// ---- Data types/Beckhoff IO udts/udt_EP2328_0002.TcDUT
(*udt (user defined type) of Beckhoff EP2028-0002 - 8 Point IP67 Rated Digital Output Box:
	auth. Brent Lekx-Toniolo of Toniolo Research & Development Inc.; 
	July 2010;
	Modified for tag reduction by R.Remillard
	November 2012; version 2.0*)


TYPE udt_EP2328_0002 :
STRUCT
	Q AT %Q*: BYTE;
	I AT %I*: BYTE;
	
	(*Status bits*)
	WC_State AT %I*:BOOL;
	State AT %I*: UINT;

END_STRUCT
END_TYPE

// ---- Data types/Beckhoff IO udts/udt_EP2624.TcDUT
(*udt (user defined type) of Beckhoff EL2624 - 4 Point Relay Type Output Terminal:
	Auth: j.vandongen
	October 2019*)


TYPE udt_EP2624 :
STRUCT
	Q: INT;
END_STRUCT
END_TYPE

// ---- Data types/Beckhoff IO udts/udt_EP2624_STAT.TcDUT
(*udt (user defined type) of Beckhoff EL2624 - 4 Point Relay Type Output Terminal:
	Auth: j.vandongen
	October 2019*)


TYPE udt_EP2624_STAT :
STRUCT
	InfoData: udt_ECATSlave_Status;
END_STRUCT
END_TYPE

// ---- Data types/Beckhoff IO udts/udt_EP3174_0002.TcDUT
(*udt (user defined type) of Beckhoff EP3174_0002 - 4 channel,  Analog Input Terminal:*)


TYPE udt_EP3174_0002 :
STRUCT

	CH1: INT;
	CH2: INT;
	CH3: INT;
	CH4: INT;
	InfoData: udt_ECATSlave_Status;

END_STRUCT
END_TYPE

// ---- Data types/Beckhoff IO udts/udt_EP6224.TcDUT
(*udt (user defined type) of Beckhoff EP6224-0002 - 4 Point IP67 Rated IO-Link Box:
	Version 20190506
		- initial creation, j.vandongen


*)


TYPE udt_EP6224 :
STRUCT

	Device_Diag: BOOL;
	Device_Stat: BOOL;


(* DeviceState Inputs:
	0x_0 = Port disabled
	0x_1 = Port in std dig in
	0x_2 = Port in std dig out
	0x_3 = Port in communikation OP
	0x_4 = Port in communikation COMSTOP
	0x1_ = Watchdog detected
	0x2_ = internal Error
	0x3_ = invalid Device ID
	0x4_ = invalid Vendor ID
	0x5_ = invalid IO-Link Version
	0x6_ = invalid Frame Capability
	0x7_ = invalid Cycle Time
	0x8_ = invalid PD in length
	0x9_ = invalid PD out length
	0xA_ = no Device detected
	0xB_ = error Preoperate
*)
	State_Ch1: USINT;
	State_Ch2: USINT;
	State_Ch3: USINT;
	State_Ch4: USINT;


	Port1_ProcessData: ARRAY [0..7] OF USINT;
	Port2_ProcessData: ARRAY [0..7] OF USINT;
	Port3_ProcessData: ARRAY [0..7] OF USINT;
	Port4_ProcessData: ARRAY [0..7] OF USINT;


	InfoData: udt_ECATSlave_StatusADS;

END_STRUCT
END_TYPE

// ---- Data types/Beckhoff IO udts/udt_EP6224_CMD.TcDUT
(*udt (user defined type) of Beckhoff EP6224-0002 - 4 Point IP67 Rated IO-Link Box:
	Version 20190506
		- initial creation, j.vandongen


*)


TYPE udt_EP6224_CMD :
STRUCT
	Port1_Q: BOOL;
	Port2_Q: BOOL;
	Port3_Q: BOOL;
	Port4_Q: BOOL;

END_STRUCT
END_TYPE

// ---- Data types/Beckhoff IO udts/udt_EP6224_I.TcDUT
(*udt (user defined type) of Beckhoff EP6224-0002 - 4 Point IP67 Rated IO-Link Box:
	Version 20210621
		- initial creation, j.underhill

*)


TYPE udt_EP6224_I :
STRUCT
	Port1_I: BOOL;
	Port2_I: BOOL;
	Port3_I: BOOL;
	Port4_I: BOOL;

END_STRUCT
END_TYPE

// ---- Data types/Beckhoff IO udts/udt_EP9128_20250704.TcDUT
(*udt (user defined type) of Beckhoff CU1128 - EtherCAT Junction:
	
------------------------------------------------------------------------
REVISION NOTES:
	Original Author(s): b.lekx-toniolo, copied from CU1128: r.jones
	Version 20250704
		- Initial Concept

------------------------------------------------------------------------
*)
TYPE udt_EP9128_20250704 :
STRUCT
	InfoData: udt_ECATSlave_Status_EP9128;
	InfoDataB: udt_ECATSlave_Status_EP9128;
	InfoDataC: udt_ECATSlave_Status_EP9128;
END_STRUCT
END_TYPE

// ---- Data types/Beckhoff IO udts/udt_EP9214_CH_CMD_20250704.TcDUT
(*udt (user defined type) of Beckhoff EP9214 IP67 Block - Power Distribution Block, individual channel data:
	To work in conjunction of udt_EP9214_STAT_yyyymmdd
	auth. Brent Lekx-Toniolo, copy/paste from 9224 from r.jones of Sodecia GTAC; 

------------------------------------------------------------------------
REVISION NOTES:
	Version 20250704
		- Initial Concept
------------------------------------------------------------------------

*)


TYPE udt_EP9214_CH_CMD_20250704 :
STRUCT

	Output_Us: BOOL;
	Output_Up: BOOL;
	Reset_Us: BOOL;
	Reset_Up: BOOL;

END_STRUCT
END_TYPE

// ---- Data types/Beckhoff IO udts/udt_EP9214_CH_STAT_20250704.TcDUT
(*udt (user defined type) of Beckhoff EP9214 IP67 Block - Power Distribution Block, individual channel data:
	To work in conjunction of udt_EP9214_STAT_yyyymmdd
	auth. Brent Lekx-Toniolo, copy/paste from 9224 from r.jones of Sodecia GTAC; 

------------------------------------------------------------------------
REVISION NOTES:
	Version 20250704
		- Initial Concept
------------------------------------------------------------------------

*)


TYPE udt_EP9214_CH_STAT_20250704 :
STRUCT

	Error_Us: BOOL;
	Error_Up: BOOL;
	Warning_Us: BOOL;
	Warning_Up: BOOL;
	Status_Us: BOOL;
	Status_Up: BOOL;
	Channel_Error: BOOL;
	SyncError: BOOL;
	TxPDO_State: BOOL;
	TxPDO_Toggle: BOOL;

END_STRUCT
END_TYPE

// ---- Data types/Beckhoff IO udts/udt_EP9214_CMD_20250704.TcDUT
(*udt (user defined type) of Beckhoff EP9214 IP67 Block - Power Distribution Block, individual channel data:
	To work in conjunction of udt_EP9214_STAT_yyyymmdd
	auth. Brent Lekx-Toniolo, copy/paste from 9224 from r.jones of Sodecia GTAC; 

------------------------------------------------------------------------
REVISION NOTES:
	Version 20250704
		- Initial Concept
------------------------------------------------------------------------
------------------------------------------------------------------------
*)
TYPE udt_EP9214_CMD_20250704 :
STRUCT

	(*Channel Specific Commands*)
	Channel1: udt_EP9214_CH_CMD_20250704;
	Channel2: udt_EP9214_CH_CMD_20250704;
	Channel3: udt_EP9214_CH_CMD_20250704;
	Channel4: udt_EP9214_CH_CMD_20250704;

	(*Overall Device Commands*)
	Device: udt_EP9214_DEV_CMD_20250704;

END_STRUCT
END_TYPE

// ---- Data types/Beckhoff IO udts/udt_EP9214_DEV_CMD_20250704.TcDUT
(*udt (user defined type) of Beckhoff EP9214 IP67 Block - Power Distribution Block, individual channel data:
	To work in conjunction of udt_EP9214_STAT_yyyymmdd
	auth. Brent Lekx-Toniolo, copy/paste from 9224 from r.jones of Sodecia GTAC; 

------------------------------------------------------------------------
REVISION NOTES:
	Version 20250704
		- Initial Concept
------------------------------------------------------------------------

*)


TYPE udt_EP9214_DEV_CMD_20250704 :
STRUCT

	Enable_Control_Via_Fieldbus: BOOL;
	Global_Reset: BOOL;

END_STRUCT
END_TYPE

// ---- Data types/Beckhoff IO udts/udt_EP9214_DEV_STAT_20250704.TcDUT
(*udt (user defined type) of Beckhoff EP9214 IP67 Block - Power Distribution Block, individual channel data:
	To work in conjunction of udt_EP9214_STAT_yyyymmdd
	auth. Brent Lekx-Toniolo, copy/paste from 9224 from r.jones of Sodecia GTAC; 

------------------------------------------------------------------------
REVISION NOTES:
	Version 20250704
		- Initial Concept
------------------------------------------------------------------------

*)


TYPE udt_EP9214_DEV_STAT_20250704 :
STRUCT

	Temperature_Warning: BOOL;
	Temperature_Error: BOOL;
	Us_Warning: BOOL;
	Us_Error: BOOL;
	Up_Warning: BOOL;
	Up_Error: BOOL;
	Global_Error_Bit: BOOL;
	Reset_Input: BOOL;
	TxPDO_State: BOOL;
	TxPDO_Toggle: BOOL;

END_STRUCT
END_TYPE

// ---- Data types/Beckhoff IO udts/udt_EP9214_STAT_20250704.TcDUT
(*udt (user defined type) of Beckhoff EP9214 IP67 Block - Power Distribution Block, individual channel data:
	To work in conjunction of udt_EP9214_STAT_yyyymmdd
	auth. Brent Lekx-Toniolo, copy/paste from 9224 from r.jones of Sodecia GTAC; 

------------------------------------------------------------------------
REVISION NOTES:
	Version 20250704
		- Initial Concept
------------------------------------------------------------------------

*)


TYPE udt_EP9214_STAT_20250704 :
STRUCT

	(*Channel Specific Status*)
	Channel_1: udt_EP9214_CH_STAT_20250704;
	Channel_2: udt_EP9214_CH_STAT_20250704;
	Channel_3: udt_EP9214_CH_STAT_20250704;
	Channel_4: udt_EP9214_CH_STAT_20250704;

	(*Overall Device Status*)
	Device: udt_EP9214_DEV_STAT_20250704;


	(*EtherCAT Slave Status*)
	Wc_State: BOOL;
	(*0 = Data valid
	1 = Data invalid*)
	InfoData: udt_ECATSlave_StatusEXT;

END_STRUCT
END_TYPE

// ---- Data types/Beckhoff IO udts/udt_EP9224_CH_CMD_20161207.TcDUT
(*udt (user defined type) of Beckhoff EP9224 IP67 Block - Power Distribution Block, individual channel commands
	To work in conjunction of udt_EP9224_CMDyymmdd
	auth. Brent Lekx-Toniolo of Sodecia GTAC; 

------------------------------------------------------------------------
REVISION NOTES:
	Version 20161207
		- Initial Concept
------------------------------------------------------------------------

*)


TYPE udt_EP9224_CH_CMD_20161207 :
STRUCT

	Output_Us: BOOL;
	Output_Up: BOOL;
	Reset_Us: BOOL;
	Reset_Up: BOOL;

END_STRUCT
END_TYPE

// ---- Data types/Beckhoff IO udts/udt_EP9224_CH_STAT_20161207.TcDUT
(*udt (user defined type) of Beckhoff EP9224 IP67 Block - Power Distribution Block, individual channel data:
	To work in conjunction of udt_EP9224_STAT_yyyymmdd
	auth. Brent Lekx-Toniolo of Sodecia GTAC; 

------------------------------------------------------------------------
REVISION NOTES:
	Version 20161207
		- Initial Concept
------------------------------------------------------------------------

*)


TYPE udt_EP9224_CH_STAT_20161207 :
STRUCT

	Error_Us: BOOL;
	Error_Up: BOOL;
	Warning_Us: BOOL;
	Warning_Up: BOOL;
	Status_Us: BOOL;
	Status_Up: BOOL;
	Channel_Error: BOOL;
	Error_Sum_Current: BOOL;
	Warning_Sum_Current: BOOL;
	TxPDO_State: BOOL;
	TxPDO_Toggle: BOOL;
	Current_Us: INT;
	Current_Up: INT;

END_STRUCT
END_TYPE

// ---- Data types/Beckhoff IO udts/udt_EP9224_CMD_20161207.TcDUT
(*udt (user defined type) of Beckhoff EP9224 IP67 Block - Power Distribution Block:
	To work in conjunction of udt_EP9224_STAT_yyyymmdd
	auth. Brent Lekx-Toniolo of Sodecia GTAC; 


------------------------------------------------------------------------
REVISION NOTES:
	Version 20161207
		- Initial Concept
------------------------------------------------------------------------
*)
TYPE udt_EP9224_CMD_20161207 :
STRUCT

	(*Channel Specific Commands*)
	Channel1: udt_EP9224_CH_CMD_20161207;
	Channel2: udt_EP9224_CH_CMD_20161207;
	Channel3: udt_EP9224_CH_CMD_20161207;
	Channel4: udt_EP9224_CH_CMD_20161207;

	(*Overall Device Commands*)
	Device: udt_EP9224_DEV_CMD_20161207;

END_STRUCT
END_TYPE

// ---- Data types/Beckhoff IO udts/udt_EP9224_DEV_CMD_20161207.TcDUT
(*udt (user defined type) of Beckhoff EP9224 IP67 Block - Power Distribution Block, device commands
	To work in conjunction of udt_EP9224_CMDyymmdd
	auth. Brent Lekx-Toniolo of Sodecia GTAC; 

------------------------------------------------------------------------
REVISION NOTES:
	Version 20161207
		- Initial Concept
------------------------------------------------------------------------

*)


TYPE udt_EP9224_DEV_CMD_20161207 :
STRUCT

	Enable_Control_Via_Fieldbus: BOOL;
	Global_Reset: BOOL;

END_STRUCT
END_TYPE

// ---- Data types/Beckhoff IO udts/udt_EP9224_DEV_STAT_20161207.TcDUT
(*udt (user defined type) of Beckhoff EP9224 IP67 Block - Power Distribution Block, device data:
	To work in conjunction of udt_EP9224_STAT_yyyymmdd
	auth. Brent Lekx-Toniolo of Sodecia GTAC; 

------------------------------------------------------------------------
REVISION NOTES:
	Version 20161207
		- Initial Concept
------------------------------------------------------------------------

*)


TYPE udt_EP9224_DEV_STAT_20161207 :
STRUCT

	Temperature_Warning: BOOL;
	Temperature_Error: BOOL;
	Us_Warning: BOOL;
	Us_Error: BOOL;
	Up_Warning: BOOL;
	Up_Error: BOOL;
	Global_Error_Bit: BOOL;
	Sum_Curent_Warning: BOOL;
	Sum_Current_Error: BOOL;
	Reset_Input: BOOL;
	TxPDO_State: BOOL;
	TxPDO_Toggle: BOOL;
	Current_Us: INT;
	Current_Up: INT;
	Voltage_Us: INT;
	Voltage_Up: INT;
	Temperature: INT;

END_STRUCT
END_TYPE

// ---- Data types/Beckhoff IO udts/udt_EP9224_STAT_20161207.TcDUT
(*udt (user defined type) of Beckhoff EP9224 IP67 Block - Power Distribution Block:
	To work in conjunction of udt_EP9224_yyyymmdd
	auth. Brent Lekx-Toniolo of Sodecia GTAC; 

------------------------------------------------------------------------
REVISION NOTES:
	Version 20161207
		- Initial Concept
------------------------------------------------------------------------

*)


TYPE udt_EP9224_STAT_20161207 :
STRUCT

	(*Channel Specific Status*)
	Channel_1: udt_EP9224_CH_STAT_20161207;
	Channel_2: udt_EP9224_CH_STAT_20161207;
	Channel_3: udt_EP9224_CH_STAT_20161207;
	Channel_4: udt_EP9224_CH_STAT_20161207;

	(*Overall Device Status*)
	Device: udt_EP9224_DEV_STAT_20161207;


	(*EtherCAT Slave Status*)
	Wc_State: BOOL;
	(*0 = Data valid
	1 = Data invalid*)
	InfoData: udt_ECATSlave_StatusEXT;

END_STRUCT
END_TYPE

// ---- Data types/Beckhoff IO udts/udt_ProfiMaster_Status.TcDUT
(*udt (user defined type) of Generic Profibus Master to Store Data for Status of any Profibus Master Modules:
	auth. brent lekx-toniolo; April 2008*)

TYPE udt_ProfiMaster_Status :
	STRUCT
		(*CdlInfo*)
		cycleCounter: UINT;
		error: USINT;
		actualCycleTime: UINT;
		actualModulo: USINT;
		(*CycleCounter:
  			FCxxxx increments this counter once after each cycle
		Error:
  			indicates the number of boxes with a BoxState unequal zero
		ActualCycleTime:
  			indicates the actual Cycle-Time (in 4/25 µs)
		ActualModulo:
  			indicates the actual Modulo in case of different poll cycles of the boxes*)

		(*Counter*)
		Counter0: UINT;
		Counter1: UINT;
		Counter2: UINT;
		Counter3: UINT;
		Counter4: UINT;
		Counter5: UINT;
		Counter6: UINT;
		Counter7: UINT;
		(*	Counter[0-1]: reserved for future
			Counter[2]: ReceivedTelegram-Counter (in Redundancy Mode)
  				FCxxxx increments this counter once every time when a correct
  				PROFIBUS-telegram is received (only in Redundancy Mode)
			Counter[3]: ReceivedTelegramFromPrimaryMaster-Counter (in Redundancy Mode)
  				FCxxxx increments this counter once every time when a correct
  				PROFIBUS-telegram from the Primary Master (which has the same
  				station address as the Redundancy Master is received (only in Redundancy Mode)
			Counter[4]: ClaimTokenTimeout-Counter (in Redundancy Mode)
  				FCxxxx increments this counter once every time when a Timeout on the
  				PROFIBUS occurs (only in Redundancy Mode)
			Counter[5-7]: reserved for future*)

		DiagFlag: BOOL;

		(*GlobalState*)
		GlobalState0: UINT;
		GlobalState1: UINT;
		GlobalState2: UINT;
		GlobalState3: UINT;
			(*GlobalState[0]:
  				0: FC310x is in state RUN
  				1: FC310x is in state RESET
  				2: FC310x is in state OFFLINE
  				3: FC310x is in state STOP
			GlobalState[1]:
  				number of bus errors detected
			GlobalState[2]:
  				reserved for future use*)

		LastAdsError: UINT;
		CycleFailedCounter: UINT;
	END_STRUCT

END_TYPE

// ---- Data types/Beckhoff IO udts/udt_ProfiNet_Status.TcDUT
TYPE udt_ProfiNet_Status :
STRUCT
	
	PnIoBoxState : UINT;
(*
0 = No error
1 = Profinet device state machine is in boot mode
2 = Device not found
3 = The stationname is not unique
4 = IP could not be set
5 = IP conflict
6 = DCP set was not successful
7 = Watchdog error
8 = Datahold error
9 = RTC3: Sync mode could not be initiated
10 = Profinet controller has a link error
11 = The aliasname is not unique
12 = The automatic name assignement isn't possible - wrong device type
13 = IOC-AR is established but no application ready
14 = IOC-AR is established but module difference
15 = At least one InputCR is invalid, provider in stop or problemindicator is set
16 = At least one OutputCR is invalid, provider in stop or problemindicator is set
31 = Only for EtherCAT gateways: WC-State of cyclic EtherCAT frame is 1
*)

END_STRUCT
END_TYPE

// ---- Data types/Beckhoff IO udts/udt_ProfiNode_Status.TcDUT
(*udt (user data type) of Generic Profibus Node to Store Data for Status of any Profibus Modules:
	auth. brent lekx-toniolo; April 2008
	version 1.0*)


TYPE udt_ProfiNode_Status :
	STRUCT
		DpState: USINT;
		(*0 = No error
		1 = Station deactivated
		2 = Station not exists
		3 = Master lock
		4 = Invalid slave response
		5 = Parameter fault
		6 = Not supported
		7 = Config fault
		8 = Station not ready
		9 = Static diagnosis
		10 = Diagnosis overflow
		11 = Physical fault
		12 = Data-Exchange left
		13 = Severe bus fault
		14 = Telegram fault
		15 = Station has no ressources
		16 = Service not activated
		17 = Unexpected telegram
		18 = Station ready
		128 = slave, waiting for data transfer
		129	= slave, waiting for configuration
		130	= slave, waiting for parameter*)
		ExtDiagFlag: BOOL;

	END_STRUCT
END_TYPE

// ---- Data types/Beckhoff IO udts/udt_SMB_Status_20141211.TcDUT
(*udt used to create memory space for linking to SMB diagnositcs
For use with Motherboards that contain LM75 and/or LM78 chips accessed via System Management Bus (SMB)


------------------------------------------------------------------------
REVISION NOTES:
	Original Author(s): b.lekx-toniolo, JVD, Chris Timmermans (Edge)
	Version 20141211
		- First Draft

------------------------------------------------------------------------
*)




TYPE udt_SMB_Status_20141211 :
STRUCT
	Temp_MB: 	UINT; 		(*°C*)
	Fan_0: 		UINT;		(*RPM*)
	Fan_1: 		UINT;		(*RPM*)
	Fan_2: 		UINT;		(*RPM*)
	Volt_2a: 		UINT;		(*0.01V*)
	Volt_2b: 		UINT;		(*0.01V*)
	Volt_33: 		UINT;		(*0.01V*)
	Volt_5: 		UINT;		(*0.01V*)
	Volt_12: 		UINT;		(*0.01V*)
	Volt_neg12: 	UINT;		(*0.01V*)
	Volt_neg5: 	UINT;		(*0.01V*)
	Temp_0: 	USINT;		(*°C*)
	Temp_1: 	USINT;		(*°C*)
	Temp_2: 	USINT;		(*°C*)
	Temp_3: 	USINT;		(*°C*)
	Temp_4: 	USINT;		(*°C*)
	Temp_5: 	USINT;		(*°C*)
	Temp_6:		USINT;		(*°C*)
	Temp_7: 	USINT;		(*°C*)


END_STRUCT
END_TYPE

// ---- Data types/Discrete Image udts/udt_ATIxx_Image_20151104.TcDUT
(*udt (user defined type) for all generic ATI Tool changers
	auth. Brent Lekx-Toniolo of Sodecia GTAC

------------------------------------------------------------------------
REVISION NOTES:

	Version 20151104:
	- initial concept, b.lekx-toniolo	
------------------------------------------------------------------------

*)

TYPE udt_ATIxx_Image_20151104 :
	STRUCT
			(*Input Data Image*)
			In_From_Hardware: udt_ATI_Input_20150203;
			(*Output Data Image*)
			Out_To_Hardware: udt_ATI_Output_20150203;

			(*Cable Break States*)
			ECatSlave_Cable_Breaks: UDINT;

	END_STRUCT
END_TYPE

// ---- Data types/Discrete Image udts/udt_Drive_Image_20160804.TcDUT
(*udt (user defined type) of Beckhoff Type for Storage of Visualization for Servo Drive Data
	auth. Brent Lekx-Toniolo of Toniolo Research & Development Inc.; 
	SORT OF RUSHED!!!
	Sept 2010; version 1.0

	Version 1.0: Sept2010
		- Initial Concept
	Version 1.1
		- A little less RUSHED, r.remillard
	Version 1.2
		- Added extra var for error April 21 2015 Chris Timmermans
	Version20160804
		- Changed Name for convention, b.lekx-toniolo
		- Moved Safety Diag and Safety Status Words from UI section to this udt, b.lekx-toniolo
		- Created Arrays for Multi axis use per drive system, b.lekx-toniolo
		- Added Seperated Error IDs and Strings, b.lekx-toniolo
*)



TYPE udt_Drive_Image_20160804 :
	STRUCT
	(*General Status of Drive SYSTEM and FB*)
	In_Play_ACK: ARRAY[1..2] OF BOOL;
	In_Teach_ACK: ARRAY[1..2] OF BOOL;
	Homed: ARRAY[1..2] OF BOOL;
	In_Motion: ARRAY[1..2] OF BOOL;
	In_Requested_Position: ARRAY[1..2] OF BOOL;
	Current_Step_Pointer: ARRAY[1..2] OF UDINT;
	At_Current_Step: ARRAY[1..2] OF UINT;
	Prev_Step_Data: ARRAY[1..2] OF udt_SingleAxis_MoveData_20160908;
	Current_Step_Data: ARRAY[1..2] OF udt_SingleAxis_MoveData_20160908;
	Next_Step_Data: ARRAY[1..2] OF udt_SingleAxis_MoveData_20160908;
	Cycle_Complete: ARRAY[1..2] OF BOOL;

	(*Status of Physical Drive Unit and Axis*)
	AX5xxx: udt_AX5206_20160804;
	EL7xxx: udt_EL7211_20150115;

	AX5805: udt_AX5805_20160804;
	Safety_DIAG: 	udt_AX5805_DiagData;
	Safety_STAT: DINT;

	Drive_Type_Message: ARRAY[1..2] OF STRING;
	Drive_OperationalState: ARRAY[1..2] OF E_AX5000_DriveOpMode;

	Drive_In_Error: ARRAY[1..2] OF BOOL;
	Drive_Status: ARRAY[1..2] OF UINT;
	Drive_StatusStruct: ARRAY[1..2] OF ST_AX5000DriveStatus;
	Drive_Status_Message: ARRAY[1..2] OF STRING;
	Drive_Diag_ErrorID: ARRAY[1..2] OF UDINT;
	Drive_Diag_Message: ARRAY[1..2] OF STRING;
	Drive_C1D_ErrorID: ARRAY[1..2] OF UINT;
	Drive_C1D_ErrorStruct: ARRAY [1..2] OF ST_AX5000_C1D;
	Drive_C1D_Error_Message: ARRAY[1..2] OF STRING;

	Axis_Motor_Message: ARRAY[1..2] OF STRING;
	Axis_In_Error: ARRAY[1..2] OF BOOL;
	Axis_ErrorID: ARRAY[1..2] OF DWORD;
	Axis_ErrorMessage: ARRAY[1..2] OF STRING;

	Actual_Position: ARRAY[1..2] OF LREAL;
	Software_Limit_Exceeded: ARRAY[1..2]OF BOOL;
	Is_Calibrated: ARRAY[1..2] OF BOOL;
	StateDWord: ARRAY[1..2] OF DWORD;
	Ready: ARRAY[1..2] OF BOOL;



	END_STRUCT
END_TYPE

// ---- Data types/Discrete Image udts/udt_Drive_Image_20190816.TcDUT
(*udt (user defined type) of Beckhoff Type for Storage of Visualization for Servo Drive Data
	auth. Brent Lekx-Toniolo of Toniolo Research & Development Inc.; 
	SORT OF RUSHED!!!
	Sept 2010; version 1.0

	Version 1.0: Sept2010
		- Initial Concept
	Version 1.1
		- A little less RUSHED, r.remillard
	Version 1.2
		- Added extra var for error April 21 2015 Chris Timmermans
	Version20160804
		- Changed Name for convention, b.lekx-toniolo
		- Moved Safety Diag and Safety Status Words from UI section to this udt, b.lekx-toniolo
		- Created Arrays for Multi axis use per drive system, b.lekx-toniolo
		- Added Seperated Error IDs and Strings, b.lekx-toniolo
		- Added Axis ID Strings, b.lekx-toniolo
	Version 20180801
		- teach enabled added, b.donnell 
	Version 20190816
		-added "Corrected Positon" var for crankshaft/coupling conversions for UI displaying purposes, j.underhill (Fork Drilling Machine)
*)



TYPE udt_Drive_Image_20190816 :
	STRUCT

	(*Identification String for general purpose UI*)
	Axis_Common_Name: ARRAY[0..2] OF STRING[30];

	(*General Status of Drive SYSTEM and FB*)
	In_Play_ACK: ARRAY[0..2] OF BOOL;
	In_Teach_ACK: ARRAY[0..2] OF BOOL;
	Homed: ARRAY[0..2] OF BOOL;
	In_Motion: ARRAY[0..2] OF BOOL;
	In_Requested_Position: ARRAY[0..2] OF BOOL;
	Current_Step_Pointer: ARRAY[0..2] OF UDINT;
	At_Current_Step: ARRAY[0..2] OF UINT;
	Prev_Step_Data: ARRAY[0..2] OF udt_SingleAxis_MoveData_20160908;
	Current_Step_Data: ARRAY[0..2] OF udt_SingleAxis_MoveData_20160908;
	Next_Step_Data: ARRAY[0..2] OF udt_SingleAxis_MoveData_20160908;
	Cycle_Complete: ARRAY[0..2] OF BOOL;
	Teach_Enable: ARRAY[0..2] OF BOOL;

	(*Status of Physical Drive Unit and Axis*)
	AX5xxx: udt_AX5206_20160804;
	EL7xxx: udt_EL7211_20150115;

	AX5805: udt_AX5805_20160804;
	Safety_DIAG: 	udt_AX5805_DiagData;
	Safety_STAT: DINT;

	Drive_Type_Message: ARRAY[0..2] OF STRING;
	Drive_OperationalState: ARRAY[0..2] OF E_AX5000_DriveOpMode;

	Drive_In_Error: ARRAY[0..2] OF BOOL;
	Drive_Status: ARRAY[0..2] OF UINT;
	Drive_StatusStruct: ARRAY[0..2] OF ST_AX5000DriveStatus;
	Drive_Status_Message: ARRAY[0..2] OF STRING;
	Drive_Diag_ErrorID: ARRAY[0..2] OF UDINT;
	Drive_Diag_Message: ARRAY[0..2] OF STRING;
	Drive_C1D_ErrorID: ARRAY[0..2] OF UINT;
	Drive_C1D_ErrorStruct: ARRAY [0..2] OF ST_AX5000_C1D;
	Drive_C1D_Error_Message: ARRAY[0..2] OF STRING;

	Axis_Motor_Message: ARRAY[0..2] OF STRING;
	Axis_In_Error: ARRAY[0..2] OF BOOL;
	Axis_ErrorID: ARRAY[0..2] OF DWORD;
	Axis_ErrorMessage: ARRAY[0..2] OF STRING;

	Corrected_Position: ARRAY[0..2] OF LREAL;
	Actual_Position: ARRAY[0..2] OF LREAL;
	Software_Limit_Exceeded: ARRAY[0..2]OF BOOL;
	Is_Calibrated: ARRAY[0..2] OF BOOL;
	StateDWord: ARRAY[0..2] OF DWORD;
	Ready: ARRAY[0..2] OF BOOL;



	END_STRUCT
END_TYPE

// ---- Data types/Discrete Image udts/udt_ECATMaster_Image_20220224.TcDUT
(*udt (user defined type) for full display (By GTAC Standards) of EtherCAT Master:
	auth. Brent Lekx-Toniolo of Toniolo Research & Development Inc.; 
	Version 20160407
		- initial concept, b.lekx-toniolo
	Version 20220224
	- Change Config array start element from 1 to 0 for TcUI migration project, b.lekx-toniolo / c.drees

*)



TYPE udt_ECATMaster_Image_20220224 :
STRUCT
	HW: udt_ECATMaster_Status_20141211;
	AMS_ID: STRING;
	Config: ARRAY [0..100] OF STRING[5];


END_STRUCT
END_TYPE

// ---- Data types/Discrete Image udts/udt_ECATNodeConfig_20200729.TcDUT
TYPE udt_ECATNodeConfig_20200729 :
STRUCT
		FixtureConfig:ARRAY [0..120] OF udt_ECATNodeData_20221507;								(*Storage Area for Actual GTAC Fixture Device Based Config*)
		EOATConfig:ARRAY[0..15] OF udt_ECATNodeData_20221507;
		ATIConfig:ARRAY[0..5] OF udt_ECATNodeData_20221507;
		WSConfig:ARRAY[0..5] OF  udt_ECATNodeData_20221507;
		PedConfig:ARRAY[0..5] OF udt_ECATNodeData_20221507;
		ReamConfig:ARRAY[0..5] OF udt_ECATNodeData_20221507;
END_STRUCT
END_TYPE

// ---- Data types/Discrete Image udts/udt_ECATNodeData_20221507.TcDUT
TYPE udt_ECATNodeData_20221507 :
STRUCT
	NodeName:ARRAY[0..63] OF STRING;
	NodeType:ARRAY[0..63] OF STRING;
	State: ARRAY[0..63] OF UINT;
	TotalNodes:INT;
END_STRUCT
END_TYPE

// ---- Data types/Discrete Image udts/udt_ECAT_NodeImage_20200618.TcDUT
TYPE udt_ECAT_NodeImage_20200618 :
STRUCT
	sType:STRING;
	
END_STRUCT
END_TYPE

// ---- Data types/Discrete Image udts/udt_EOATxx_Image_20170607.TcDUT
(*udt (user defined type) for all generic EOAT (End of Arm Tools)
	auth. Brent Lekx-Toniolo of Sodecia GTAC

------------------------------------------------------------------------
REVISION NOTES:

	Version 20151103:
	- initial concept, b.lekx-toniolo	
	Version 20170607
	- unknown changes or editor
------------------------------------------------------------------------

*)

TYPE udt_EOATxx_Image_20170607 :
	STRUCT
			(*Input nodes*)
			N01: udt_EP1008_002_v2;
			N02: udt_EP1008_002_v2;
			N03: udt_EP1008_002_v2;
			N04: udt_EP1008_002_v2;
			N05: udt_EP1008_002_v2;
			N06: udt_EP1008_002_v2;
			N07: udt_EP1008_002_v2;
			N08: udt_EP1008_002_v2;
			N09: udt_EP1008_002_v2;

			(*Valve Bank*)
			N100: udt_SMC_EX260_ValveBank;
			N100_STAT: udt_SMC_EX260_STAT;
			(*Cable Break States*)
			ECatSlave_Cable_Breaks: ARRAY[0..1] OF DINT;
			(*Node Counts*)
			NodeLayout:udt_ECATNodeData_20221507;
			NodeState:ARRAY[0..63] OF UINT;
			Input_Node_Count: UDINT;
			Safety_Node_Count:Udint;
			VB_Node_Count: UDINT;

			
			(*Developed Data*)
			CLFaults1: UDINT;
			CLFaults2: UDINT;
			CLFaults3: UDINT;
			CLFaults4: UDINT;
			CLFaulted: UDINT;
			PPFaults: UDINT;
			PPFaulted: UDINT;
			(*ID*)
			ID: UINT;
			strID: STRING[255];

	END_STRUCT
END_TYPE

// ---- Data types/Discrete Image udts/udt_EOATxx_Image_20220715.TcDUT
(*udt (user defined type) for all generic EOAT (End of Arm Tools)
	auth. Brent Lekx-Toniolo of Sodecia GTAC

------------------------------------------------------------------------
REVISION NOTES:

	Version 20151103:
	- initial concept, b.lekx-toniolo	
	Version 20170607
	- unknown changes or editor
	Version 20220715
	-Added Node Layout for Auto Node identification
------------------------------------------------------------------------

*)

TYPE udt_EOATxx_Image_20220715 :
	STRUCT
			(*Input nodes*)
			N01: udt_EP1008_002_v2;
			N02: udt_EP1008_002_v2;
			N03: udt_EP1008_002_v2;
			N04: udt_EP1008_002_v2;
			N05: udt_EP1008_002_v2;
			N06: udt_EP1008_002_v2;
			N07: udt_EP1008_002_v2;
			N08: udt_EP1008_002_v2;
			N09: udt_EP1008_002_v2;

			(*Valve Bank*)
			N100: udt_SMC_EX260_ValveBank;
			N100_STAT: udt_SMC_EX260_STAT;
			(*Cable Break States*)
			ECatSlave_Cable_Breaks: UDINT;
			(*Node Counts*)
			NodeLayout:udt_ECATNodeData_20221507;
			Input_Node_Count: UDINT;
			VB_Node_Count: UDINT;
			Output_Node_Count:UDINT;
			
			(*Developed Data*)
			CLFaults1: UDINT;
			CLFaults2: UDINT;
			CLFaults3: UDINT;
			CLFaults4: UDINT;
			CLFaulted: UDINT;
			PPFaults: UDINT;
			PPFaulted: UDINT;
			(*ID*)
			ID: UINT;
			strID: STRING[255];

	END_STRUCT
END_TYPE

// ---- Data types/Discrete Image udts/udt_ESWxx_Image_20150814.TcDUT
(*udt (user defined type) for all generic ESW (Enabling Switch Option Plate) I/O Required
	auth. Brent Lekx-Toniolo of Sodecia GTAC

------------------------------------------------------------------------
REVISION NOTES:

	Version 20150814:
	- initial concept, b.lekx-toniolo	
------------------------------------------------------------------------

*)

TYPE udt_ESWxx_Image_20150814 :
STRUCT
			N01: 							udt_EP1908_002;

END_STRUCT
END_TYPE

// ---- Data types/Discrete Image udts/udt_FixXX_Input_Image_20180202.TcDUT
(*udt (user defined type) for all fixture input interface
	auth. Rob Remillard and Brent Lekx-Toniolo of Sodecia GTAC

------------------------------------------------------------------------
REVISION NOTES:
	V1.0 (pre date naming)
	- initial concept, r.remillard/b.lekx-toniolo
	Version 20160503:
	- added node and VB configuration variables, b.lekx-toniolo	
	Version 20170415:
	-added second set of ManReqs2, j.vandongen
	Version 20170612:
	-added third set of ManReqs3, j.vandongen
	Version 20170801:
	-added ManReqs1, j.vandongen
	Version 20180202:
	-added Output_Node_Count and Water_Stand_Count, j.vandongen
	Version 20220715:
	-Added the Data for handling Auto Fixture Layouts -C.Drees
	
------------------------------------------------------------------------

*)


TYPE udt_FixXX_Input_Image_20180202 :
STRUCT
	Mode_Select: INT;
	ResetProd: BOOL;
	ModelData: INT;
	ManReqs: DINT;
	ManReqs1: DINT;
	ManReqs2: DINT;
	ManReqs3: DINT;
	Go_Home: BOOL;
	Bypass_REQS: UDINT;
	CustomApplication_REQS: UDINT;
(*Node Counts and configuration data*)
	Input_Node_Count: UDINT;
	VB_Node_Count: UDINT;
	Output_Node_Count: UDINT;
	Water_Stand_Count: UDINT;

	(*Conveyor*)
	Manual_Conveyor_Start : BOOL;	
END_STRUCT
END_TYPE

// ---- Data types/Discrete Image udts/udt_FixXX_Output_Image_20220715.TcDUT
(*Generic Data Type For transfering I/O Data to HMI For visualization
	Version 20220715:
	-Added the Data for handling Auto Fixture Layouts, c.drees
	Edit 20250514:
	-Added "IsEnabled" control for Clamps, Quality, and Manual screen - Will. K 
	
	*)

TYPE udt_FixXX_Output_Image_20220715 :
	STRUCT
			InAuto: BOOL;
			InManual: BOOL;
			ManInds: DINT;
			ManInds2: DINT;
			ManInds3: DINT;
			At_Home: BOOL;
			All_Sensors_Off: BOOL;
			ReadyTo_Load: BOOL;
			Status: INT;
			ProdCount: INT;
			CycleTime: TIME;
			LoadTime: TIME;
			WeldTime: TIME;
			UnloadTime: TIME;
			PrevCycleTime: TIME;
			ToolID: INT;
			Model_Data: INT;
			CLFaults1: UDINT;
			CLFaults2: UDINT;
			CLFaults3: UDINT;
			CLFaults4: UDINT;
			CLFaulted: UDINT;
			PPFaults: UDINT;
			PPFaults1: UDINT;
			PPFaults2: UDINT;
			PPFaulted: UDINT;
			Enable_Motion: BOOL;
			Bypass_ACKS: UDINT;
			CustomApplication_ACKS: UDINT;
			Operator_Performance_Pen: REAL;
			Fixture_Allow_Model_Change: BOOL;

			N00: udt_EP1111;
			N01: udt_EP1008_002_v2;
			N02: udt_EP1008_002_v2;
			N03: udt_EP1008_002_v2;
			N04: udt_EP1008_002_v2;
			N05: udt_EP1008_002_v2;
			N06: udt_EP1008_002_v2;
			N07: udt_EP1008_002_v2;
			N08: udt_EP1008_002_v2;
			N09: udt_EP1008_002_v2;
			N10: udt_EP1008_002_v2;
			N11: udt_EP1008_002_v2;
			N12: udt_EP1008_002_v2;
			N13: udt_EP1008_002_v2;
			N14: udt_EP1008_002_v2;
			N15: udt_EP1008_002_v2;
			N16: udt_EP1008_002_v2;
			N17: udt_EP1008_002_v2;
			N18: udt_EP1008_002_v2;
			N19: udt_EP1008_002_v2;
			N20: udt_EP1008_002_v2;
			N21: udt_EP1008_002_v2;
			N22: udt_EP1008_002_v2;

			N70: udt_EP3174_0002;
			Water_Temp_1: REAL;
			Water_Flow_1: REAL;

			N30: udt_EP2028_002_v2;
			N30_STAT: udt_EP2028_002_STAT;

			N100: udt_SMC_EX260_ValveBank;
			N100_STAT: udt_SMC_EX260_STAT;
			N101: udt_SMC_EX260_ValveBank;
			N101_STAT: udt_SMC_EX260_STAT;
			N102: udt_SMC_EX260_ValveBank;
			N102_STAT: udt_SMC_EX260_STAT;
			(*Cable Break States*)
			ECatSlave_Cable_Breaks: ARRAY[0..1] OF DINT;
			(*Node Counts*)
			NodeLayout:udt_ECATNodeData_20221507;
			NodeState: ARRAY[0..63] OF UINT;
			Input_Node_Count: UDINT;
			Output_Node_Count:UDINT;
			Analog_Node_Count:Udint;
			VB_Node_Count: UDINT;
			VB_Screen_Position: UDINT;
			Water_Stand_Count: UDINT;
			
			(*IsEnabled control For UI screen*)
			Enable_FixtureContext_Clamps : BOOL;
			Enable_FixtureContext_QA : BOOL;
			Enable_FixtureContext_Manual : BOOL;
		
			(*Conveyor*)
			Conveyor_In_Progress : BOOL;
				

			
	END_STRUCT
END_TYPE

// ---- Data types/Discrete Image udts/udt_FixXX_Output_Image_20250721_CUSTOM.TcDUT
(*Generic Data Type For transfering I/O Data to HMI For visualization
	Version 20220715:
	-Added the Data for handling Auto Fixture Layouts, c.drees
	Version 20250721_CUSTOM:
	-Added more Fixture Nodes for Bumper project, w.griffiths
	
	*)

TYPE udt_FixXX_Output_Image_20250721_CUSTOM :
	STRUCT
			InAuto: BOOL;
			InManual: BOOL;
			ManInds: DINT;
			ManInds2: DINT;
			ManInds3: DINT;
			At_Home: BOOL;
			All_Sensors_Off: BOOL;
			ReadyTo_Load: BOOL;
			Status: INT;
			ProdCount: INT;
			CycleTime: TIME;
			LoadTime: TIME;
			WeldTime: TIME;
			UnloadTime: TIME;
			PrevCycleTime: TIME;
			ToolID: INT;
			Model_Data: INT;
			CLFaults1: UDINT;
			CLFaults2: UDINT;
			CLFaults3: UDINT;
			CLFaults4: UDINT;
			CLFaulted: UDINT;
			PPFaults: UDINT;
			PPFaults1: UDINT;
			PPFaults2: UDINT;
			PPFaulted: UDINT;
			Enable_Motion: BOOL;
			Bypass_ACKS: UDINT;
			CustomApplication_ACKS: UDINT;
			Operator_Performance_Pen: REAL;
			Fixture_Allow_Model_Change: BOOL;

			N00: udt_EP1111;
			N01: udt_EP1008_002_v2;
			N02: udt_EP1008_002_v2;
			N03: udt_EP1008_002_v2;
			N04: udt_EP1008_002_v2;
			N05: udt_EP1008_002_v2;
			N06: udt_EP1008_002_v2;
			N07: udt_EP1008_002_v2;
			N08: udt_EP1008_002_v2;
			N09: udt_EP1008_002_v2;
			N10: udt_EP1008_002_v2;
			N11: udt_EP1008_002_v2;
			N12: udt_EP1008_002_v2;
			N13: udt_EP1008_002_v2;
			N14: udt_EP1008_002_v2;
			N15: udt_EP1008_002_v2;
			N16: udt_EP1008_002_v2;
			N17: udt_EP1008_002_v2;
			N18: udt_EP1008_002_v2;
			N19: udt_EP1008_002_v2;
			N20: udt_EP1008_002_v2;
			N21: udt_EP1008_002_v2;
			N22: udt_EP1008_002_v2;
			N23: udt_EP1008_002_v2;
			N24: udt_EP1008_002_v2;
			N25: udt_EP1008_002_v2;
			N26: udt_EP1008_002_v2;
			N27: udt_EP1008_002_v2;
			N28: udt_EP1008_002_v2;
			N29: udt_EP1008_002_v2;
			N30: udt_EP1008_002_v2;
			N31: udt_EP1008_002_v2;
			N32: udt_EP1111;
			N33: udt_EP1008_002_v2;
			N34: udt_EP1111;
			N35: udt_EP1008_002_v2;
			N36: udt_EP1111;
			N37: udt_EP1008_002_v2;
			N38: udt_EP1111;
			N39: udt_EP1008_002_v2;
			N40: udt_EP1111;
			N41: udt_EP1008_002_v2;
			N42: udt_EP1111;
			N43: udt_EP1008_002_v2;

			N70: udt_EP3174_0002;
			Water_Temp_1: REAL;
			Water_Flow_1: REAL;
(*
			N30: udt_EP2028_002_v2;
			N30_STAT: udt_EP2028_002_STAT;
*)
			N100: udt_SMC_EX260_ValveBank;
			N100_STAT: udt_SMC_EX260_STAT;
			N101: udt_SMC_EX260_ValveBank;
			N101_STAT: udt_SMC_EX260_STAT;
			N102: udt_SMC_EX260_ValveBank;
			N102_STAT: udt_SMC_EX260_STAT;
			(*Cable Break States*)
			ECatSlave_Cable_Breaks: ARRAY[0..1] OF DINT;
			(*Node Counts*)
			NodeLayout:udt_ECATNodeData_20221507;
			NodeState: ARRAY[0..63] OF UINT;
			Input_Node_Count: UDINT;
			Output_Node_Count:UDINT;
			Analog_Node_Count:Udint;
			VB_Node_Count: UDINT;
			VB_Screen_Position: UDINT;
			Water_Stand_Count: UDINT;

	END_STRUCT
END_TYPE

// ---- Data types/Discrete Image udts/udt_FixXX_Persistent_Input.TcDUT
TYPE udt_FixXX_Persistent_Input :
STRUCT

	Prod_Ref_Time:						UINT;
	Prod_Target:							UINT;

END_STRUCT
END_TYPE

// ---- Data types/Discrete Image udts/udt_Fronius_Status_20170531.TcDUT
(*udt (user defined type) for all generic Fronius Type Controllers
	auth. Brent Lekx-Toniolo of Sodecia GTAC

------------------------------------------------------------------------
REVISION NOTES:

	Version 20170531:
		- initial concept, b.lekx-toniolo	


------------------------------------------------------------------------

*)



TYPE udt_Fronius_Status_20170531 :
STRUCT

	Ready: BOOL;
	Error_Code: INT;
	Weld_Voltage: UDINT;
	Weld_Current: UDINT;
	Weld_WFS: UDINT;

END_STRUCT
END_TYPE

// ---- Data types/Discrete Image udts/udt_ICxx_Image.TcDUT
(*udt (user defined type) for all generic IC (Industrial Controller) I/O Required
	auth. Brent Lekx-Toniolo of Toniolo Research & Development Inc.

------------------------------------------------------------------------
REVISION NOTES:

	Version??? (created before the begining of time):
	- initial concept, b.lekx-toniolo	
------------------------------------------------------------------------

*)
TYPE udt_ICxx_Image :
	STRUCT
		T01: udt_EK1100;					(*Ecat Bus Coupler*)
		T02_STAT: udt_EL6900_STAT_20160426;	(*EL Safety CPU*)
		T02_CMD: udt_EL6900_CMD_20121204;
		T03: udt_EL1904_v2;				(*EL Safety Inputs*)
		T04: udt_EL1904_v2;				(*EL Safety Inputs*)
		T05: udt_EL1904_v2;				(*EL Safety Inputs*)
		T06: udt_EL1904_v2;				(*EL Safety Inputs*)
		T07: udt_EL1904_v2;				(*EL Safety Inputs*)
		T08: udt_EL1904_v2;				(*EL Safety Inputs*)
		T09: udt_EL2904RO_v2;			(*EL Safety Outputs, Set to "I" as this terminal is safety rated, therefore read only!*)
		T10: udt_EL2904RO_v2;			(*EL Safety Outputs, Set to "I" as this terminal is safety rated, therefore read only!*)
		T11: udt_EL94xx;					(*EBUS Power Restoration*)
		T12: udt_EL1004_v2;				(*EL Inputs*)
		T13: udt_EL1004_v2;				(*EL Inputs*)
		T14: udt_EL2008_v2;				(*EL Outputs, 8 Point*)
		T14_STAT: udt_EL2008_STAT;		(*EL Output Card Status*)
		T15: udt_EL2622;					(*EL Outputs, 4 Point*)
		T15_STAT: udt_EL2622_STAT;		(*EL Output Card Status*)
		T16: udt_EK1122; 					(*ECAT Junction*)

	END_STRUCT
END_TYPE

// ---- Data types/Discrete Image udts/udt_ICxx_Image_20201104.TcDUT
(*udt (user defined type) for all generic IC (Industrial Controller) I/O Required
	auth. Brent Lekx-Toniolo of Toniolo Research & Development Inc.

------------------------------------------------------------------------
REVISION NOTES:

	Version??? (created before the begining of time):
	- initial concept, b.lekx-toniolo	
------------------------------------------------------------------------

*)
TYPE udt_ICxx_Image_20201104 :
	STRUCT
		T01: udt_EK1100;					(*Ecat Bus Coupler*)
		T02_STAT: udt_EL6900_STAT_20160426;	(*EL Safety CPU*)
		T02_CMD: udt_EL6900_CMD_20121204;
		T03: udt_EL1904_v2;				(*EL Safety Inputs*)
		T04: udt_EL1904_v2;				(*EL Safety Inputs*)
		T05: udt_EL1904_v2;				(*EL Safety Inputs*)
		T06: udt_EL1904_v2;				(*EL Safety Inputs*)
		T07: udt_EL1904_v2;				(*EL Safety Inputs*)
		T08: udt_EL1904_v2;				(*EL Safety Inputs*)
		T09: udt_EL2904RO_v2;			(*EL Safety Outputs, Set to "I" as this terminal is safety rated, therefore read only!*)
		T10: udt_EL2904RO_v2;			(*EL Safety Outputs, Set to "I" as this terminal is safety rated, therefore read only!*)
		T11: udt_EL94xx;					(*EBUS Power Restoration*)
		T12: udt_EL1004_v2;				(*EL Inputs*)
		T13: udt_EL1004_v2;				(*EL Inputs*)
		T14: udt_EL2008_v2;				(*EL Outputs, 8 Point*)
		T14_STAT: udt_EL2008_STAT;		(*EL Output Card Status*)
		T15: udt_EL2622;					(*EL Outputs, 4 Point*)
		T15_STAT: udt_EL2622_STAT;		(*EL Output Card Status*)
		T16: udt_EK1122; 					(*ECAT Junction*)

	END_STRUCT
END_TYPE

// ---- Data types/Discrete Image udts/udt_MDxx_Image_20251008.TcDUT
(*udt (user defined type) for all Rite Hite I-Comm Models

------------------------------------------------------------------------
REVISION NOTES:

	Version 20230719:
	- Original Concept, a. lopez
	Version 20251008:
	- Revamp per Hardware Design requests, b.lekx-toniolo
	
------------------------------------------------------------------------
*)


TYPE udt_MDxx_Image_20251008 :
	STRUCT
	
	N01_STAT: udt_EP1918_STAT_20250213;					(*EP Twinsafe*)
	N02: udt_EP1008_002_v2;								(*EP Inputs*)
	N03: udt_EP2624;									(*EP 4ch Relay Output*)
	N03_STAT: udt_EP2624_STAT;							(*EP 4ch Relay Output Card Status*)

	END_STRUCT
END_TYPE

// ---- Data types/Discrete Image udts/udt_NutWeldLVDT_Input_Image_20250616.TcDUT
(*udt (user defined type) for all Nut Weld based LVDT applications UI input interface (non presistant inputs)
	auth. Brent Lekx-Toniolo of Sodecia GTAC

------------------------------------------------------------------------
REVISION NOTES:
	Version 20250616:
	- initial concept, b.lekx-toniolo
------------------------------------------------------------------------

*)


TYPE udt_NutWeldLVDT_Input_Image_20250616 :
STRUCT
	Nut_Retry_REQ: BOOL;
	Save_LVDT_REQ: BOOL;
	Save_Nut_REQ: BOOL;
	UpperElectrode_Reset: BOOL;
END_STRUCT
END_TYPE

// ---- Data types/Discrete Image udts/udt_NutWeldLVDT_Output_Image_20250616.TcDUT
(*udt (user defined type) for all Nut Weld based LVDT applications UI ouput interface
	auth. Brent Lekx-Toniolo of Sodecia GTAC

------------------------------------------------------------------------
REVISION NOTES:
	Version 20250616:
	- initial concept, b.lekx-toniolo
------------------------------------------------------------------------

*)



TYPE udt_NutWeldLVDT_Output_Image_20250616 :
STRUCT
	LVDT_Saved_ACK: BOOL;
	Nut_Saved_ACK: BOOL;
	LVDT_Value_Raw: REAL;
	LVDT_Value_Scaled: REAL;
	LVDT_Nut_OK: BOOL;
	LVDT_Pin_ADVD: BOOL;
	LVDT_Pin_RETD: BOOL;
	
	UpperElectrode_WeldCount: UINT;	
END_STRUCT
END_TYPE

// ---- Data types/Discrete Image udts/udt_NWx_Image.TcDUT
TYPE udt_NWx_Image :
STRUCT
			InAuto: BOOL;
			InManual: BOOL;
			ManInds: DINT;
			At_Home: BOOL;
			All_Sensors_Off: BOOL;
			ReadyTo_Load: BOOL;
			Status: INT;
			ProdCount: INT;
			CycleTime: TIME;
			LoadTime: TIME;
			WeldTime: TIME;
			UnloadTime: TIME;
			PrevCycleTime: TIME;
			ToolID: INT;
			Model_Data: INT;
			CLFaults: UDINT;
			CLFaults2: UDINT;
			CLFaults3: UDINT;
			CLFaults4: UDINT;
			CLFaulted: UDINT;
			PPFaults: UDINT;
			PPFaulted: UDINT;
			Enable_Motion: BOOL;
			Weld_Curtain_Is_Bypassed: BOOL;
			Vacuum_Is_Bypassed: BOOL;
			Marker_Running: BOOL;
			Marker_Com_OK: BOOL;
			Marker_Is_Bypassed: BOOL;
			Marker_Start_Signal_Monitor: BOOL;
			Marker_Complete: BOOL;


			T01: 				udt_EK1100;
			T02_STAT: 			udt_EL6900_STAT_20160426;		(*EL Safety CPU*)
			T02_CMD: 			udt_EL6900_CMD_20121204;
			T03: 				udt_EL1904_v2;
			T04: 				udt_EL2904RO_v2;				(*Set to "I" as this terminal is safety rated, therefore read only!*)
			T05: 				udt_EL1004_v2;
			T15: 				udt_EL2622;						(*EL Outputs, 4 Point*)
			T15_STAT: 			udt_EL2622_STAT;				(*EL Output Card Status*)

END_STRUCT
END_TYPE

// ---- Data types/Discrete Image udts/udt_ISxx_Image_20241121.TcDUT
(*udt (user defined type) for all generic PD (Power Distribution Cabinet) I/O Required
	auth. Brent Lekx-Toniolo of Sodecia GTAC

------------------------------------------------------------------------
REVISION NOTES:

	Version 20150812:
		- initial concept, b.lekx-toniolo	
	Version 20170307
		- added area for N999, b.lexk-toniolo
		- added Option vars to pass data for UI config automation, b.lekx-toniolo
	Version 20190924
		- changed T05 to EL6731, moved EK1110 to T06, j.vandongen
		- added Option input for EL6731, j.vandongen
	Version 20220907
		-Added N1000 and N1001 variables for additional EP9224, C.Drees
	Version 20241121
		-PD to IS rename, as per GH SSCC610 repo Issue#162, b.lekx-toniolo		
------------------------------------------------------------------------

*)

TYPE udt_ISxx_Image_20241121 :
	STRUCT
		T01: udt_EK1100;						(*Ecat Bus Coupler*)
		T02_STAT: udt_EL6900_STAT_20160426;	(*EL Safety CPU*)
		T02_CMD: udt_EL6900_CMD_20121204;
		T03: udt_EL1904_v2;					(*EL Safety Inputs*)
		T04: udt_EL2904RO_v2;				(*EL Safety Outputs, Set to "I" as this terminal is safety rated, therefore read only!*)
		T05: udt_EL6731;						(*EL Profibus Master*)
		T06: udt_EK1110_20150812;				(*Ecat Extension Terminal*)

		N01: udt_CU1128_20180507;			(*Ecat Junction Switch*)

		N999_STAT: udt_EP9224_STAT_20161207;	(*EP Power Distribution Box*)
		N999_CMD: udt_EP9224_CMD_20161207;
		N1000_STAT: udt_EP9224_STAT_20161207;
		N1000_CMD:udt_EP9224_CMD_20161207;
		N1001_STAT:udt_EP9224_STAT_20161207;
		N1001_CMD:udt_EP9224_CMD_20161207;
		
		Option_Enable_SplitRelays: BOOL;
		Option_EP9224_Count: Int;
		Option_Enable_Pbus: BOOL;



	END_STRUCT
END_TYPE

// ---- Data types/Discrete Image udts/udt_PEDxx_Image_20170725.TcDUT
(*udt (user defined type) for all generic PEDs (Pedastals)
	auth. Brent Lekx-Toniolo of Sodecia GTAC

------------------------------------------------------------------------
REVISION NOTES:

	Version 20151104:
	- initial concept, b.lekx-toniolo	
	Version 20170725:
	- added PP faults, j.vandongen
	- added means of hiding N100 on the UI, j.vandongen
------------------------------------------------------------------------

*)

TYPE udt_PEDxx_Image_20170725 :
	STRUCT


			(*Input nodes*)
			N01: udt_EP1008_002_v2;
			N02: udt_EP1008_002_v2;

			(*Valve Bank*)
			N100: udt_SMC_EX260_ValveBank;
			N100_STAT: udt_SMC_EX260_STAT;

			(*Cable Break States*)
			ECatSlave_Cable_Breaks: UDINT;

			(*Developed Data*)
			CLFaults1: UDINT;
			CLFaults2: UDINT;
			CLFaults3: UDINT;
			CLFaults4: UDINT;
			CLFaulted: UDINT;
			PPFaults: UDINT;
			PPFaulted: UDINT;

			VB_Node_Count: UDINT;

	END_STRUCT
END_TYPE

// ---- Data types/Discrete Image udts/udt_PEDxx_Image_20240808.TcDUT
(*udt (user defined type) for all generic PEDs (Pedastals)
	auth. Brent Lekx-Toniolo of Sodecia GTAC

------------------------------------------------------------------------
REVISION NOTES:

	Version 20151104:
	- initial concept, b.lekx-toniolo	
	Version 20170725:
	- added PP faults, j.vandongen
	- added means of hiding N100 on the UI, j.vandongen
	Version 20191115
	- added N50, j.vandongen
	Version 20240514
	- added in Ped Type and Node Layout for future addition ideas, b.lekx-toniolo
	Version 20240808
	- added in the option variables for UI auto configuration, b.lekx-toniolo
------------------------------------------------------------------------

*)

TYPE udt_PEDxx_Image_20240808 :
	STRUCT

			(*Ped Type*)
			Ped_Type: INT;
	
			(*Input nodes*)
			N01: udt_EP1008_002_v2;
			N02: udt_EP1008_002_v2;

			(*Output nodes*)
			N50: udt_EP2028_002_v2;
			N50_STAT: udt_EP2028_002_STAT;

			(*Valve Bank*)
			N100: udt_SMC_EX260_ValveBank;
			N100_STAT: udt_SMC_EX260_STAT;

			(*Cable Break States*)
			ECatSlave_Cable_Breaks: ARRAY[0..1] OF DINT;

			(*Developed Data*)
			CLFaults1: UDINT;
			CLFaults2: UDINT;
			CLFaults3: UDINT;
			CLFaults4: UDINT;
			CLFaulted: UDINT;
			PPFaults: UDINT;
			PPFaulted: UDINT;
			NodeLayout:udt_ECATNodeData_20221507;

			Input_Node_Count: UDINT;
			Output_Node_Count: UDINT;
			VB_Node_Count: UDINT;
			Option_SwingCylinder: BOOL;		
			Option_TipDresser: BOOL;	
			Option_TipChanger: BOOL;	
			Part_Present_Count: UDINT;

	END_STRUCT
END_TYPE

// ---- Data types/Discrete Image udts/udt_Reamerxx_Image_20180405.TcDUT
(*udt (user defined type) for all generic Reamers (Mig Weld Tip Reamers)
	auth. Brent Lekx-Toniolo of Sodecia GTAC

------------------------------------------------------------------------
REVISION NOTES:

	Version 20160210:
	- initial concept, b.lekx-toniolo	
	Version 20180405
	- changed N20 to N30 to follow standards, j.vandongen
------------------------------------------------------------------------

*)

TYPE udt_Reamerxx_Image_20180405 :
	STRUCT
			(*Input nodes*)
			N01: udt_EP1008_002_v2;

			(*Output nodes*)
			N30: udt_EP2028_002_v2;
			N30_STAT: udt_EP2028_002_STAT;

			(*Cable Break States*)
			ECatSlave_Cable_Breaks: UDINT;

	END_STRUCT
END_TYPE

// ---- Data types/Discrete Image udts/udt_RobotDiscreteNode_Image.TcDUT
TYPE udt_RobotDiscreteNode_Image :
	STRUCT
		T01: udt_EK1100;				(*Ecat Bus Coupler*)
		(*T02_STAT: udt_EL6900_STAT;	(*EL Safety CPU*)
		T02_CMD: udt_EL6900_CMD;*)
		T03: udt_EL1904;				(*EL Safety Inputs*)
		T04: udt_EL1904;				(*EL Safety Inputs*)
		T05: udt_EL1904;				(*EL Safety Inputs*)
		T06: udt_EL1904;				(*EL Safety Inputs*)
		T07: udt_EL1904;				(*EL Safety Inputs*)
		T08: udt_EL2904RO;			(*EL Safety Outputs, Set to "I" as this terminal is safety rated, therefore read only!*)
		T09: udt_EL2904RO; 			(*EL Safety Outputs, Set to "I" as this terminal is safety rated, therefore read only!*)
		T10: udt_EL94xx;				(*EBUS Power Restoration*)
		T11: udt_EL1004;				(*EL Inputs*)
		T12: udt_EL2622;				(*EL Outpus*)
		T12_STAT: udt_EL2622_STAT;	(*EL Output Card Status*)
		T13: udt_EL1004;				(*EL Inputs, TO BE REPLACED WITH ANALOG CARD PENDING DELIVERY*)
		T14: udt_EL6731;				(*EL Profibus Mater Terminal*)

	END_STRUCT
END_TYPE

// ---- Data types/Discrete Image udts/udt_RobotDiscreteNode_ImageFSOE_20151028.TcDUT
(*udt (user defined type) for Visualization of Robot Discrete Image Conforming to SSCCV5.00 with SAFEOP + FSoE (Kuka)
	Author(S): Brent Lekx-Toniolo;
	Version 20151028
		- Initial Concept,blt

*)
TYPE udt_RobotDiscreteNode_ImageFSOE_20151028 :
	STRUCT

		T01: udt_EK1100;						(*Ecat Bus Coupler*)
		T02_STAT: udt_EL6900_STAT_20160426;	(*EL Safety CPU*)
		T02_CMD: udt_EL6900_CMD_20121204;
		T03 : udt_EL1904_v2;					(*EL1904*)
		T04: udt_EK1122;						(*EK1122*)

		RT01: udt_EK1100;					(*EK1100 for SYS-X-44 master connection*)
		RT02: udt_EL6695_20151028;			(*EL EtherCat Bridge, Specific to Kuka FSOE*)

	END_STRUCT
END_TYPE

// ---- Data types/Discrete Image udts/udt_RobotDiscreteNode_ImageSSCCv46wSAFEOP_20131903.TcDUT
(*udt (user defined type) for Visualization of Robot Discrete Image Conforming to SSCCv4.6 with SAFEOP (Kuka)
	Author(S): Brent Lekx-Toniolo/Rob Remillard of Sodecia GTAC;
	Version 20131903
		- Initial Concept

	Last Edit: March 19th, 2013, blt
		- Updated per V4.6 hardware changes
*)
TYPE udt_RobotDiscreteNode_ImageSSCCv46wSAFEOP_20131903 :
	STRUCT

		T01: udt_EK1100;				(*Ecat Bus Coupler*)
		T02_STAT: udt_EL6900_STAT_20160426;	(*EL Safety CPU*)
		T02_CMD: udt_EL6900_CMD_20121204;
		T03: udt_EL1904_v2;				(*EL Safety Inputs*)
		T04: udt_EL1904_v2;				(*EL Safety Inputs*)
		T05: udt_EL1904_v2;				(*EL Safety Inputs*)
		T06: udt_EL1904_v2;				(*EL Safety Inputs*)
		T07: udt_EL1904_v2;				(*EL Safety Inputs*)
		T08: udt_EL2904RO_v2;			(*EL Safety Outputs, Set to "I" as this terminal is safety rated, therefore read only!*)
		T09: udt_EL2904RO_v2; 			(*EL Safety Outputs, Set to "I" as this terminal is safety rated, therefore read only!*)
		T10: udt_EL6692_20121204;			(*EL EtherCat Bridge*)

	END_STRUCT
END_TYPE

// ---- Data types/Discrete Image udts/udt_RobotDiscreteNode_ImageSSCCv46_20121204.TcDUT

(*udt (user defined type) for Visualization of Robot Discrete Image Conforming to SSCCv4.6
	Author(S): Brent Lekx-Toniolo/Rob Remillard of Sodecia GTAC;
	Version 20121204
		- Intiial Concept

	Last Edit: December 5th, 2012, blt
		- Added Slave State Message Variables

*)

TYPE udt_RobotDiscreteNode_ImageSSCCv46_20121204 :
	STRUCT
		T01: udt_EK1100;				(*Ecat Bus Coupler*)
		T02_STAT: udt_EL6900_STAT_20160426;	(*EL Safety CPU*)
		T02_CMD: udt_EL6900_CMD_20121204;
		T03: udt_EL1904_v2;				(*EL Safety Inputs*)
		T04: udt_EL1904_v2;				(*EL Safety Inputs*)
		T05: udt_EL1904_v2;				(*EL Safety Inputs*)
		T06: udt_EL1904_v2;				(*EL Safety Inputs*)
		T07: udt_EL1904_v2;				(*EL Safety Inputs*)
		T08: udt_EL2904RO_v2;			(*EL Safety Outputs, Set to "I" as this terminal is safety rated, therefore read only!*)
		T09: udt_EL2904RO_v2; 			(*EL Safety Outputs, Set to "I" as this terminal is safety rated, therefore read only!*)
		T10: udt_EL6731;				(*EL Profibus Mater Terminal*)
	END_STRUCT
END_TYPE

// ---- Data types/Discrete Image udts/udt_RobotDiscreteNode_ImageSSCCv46_20131001.TcDUT
(*udt (user defined type) for Visualization of Robot Discrete Image Conforming to SSCCv4.6
	Author(S): Brent Lekx-Toniolo/Rob Remillard of Sodecia GTAC;
	Version 20121204
		- Intiial Concept

	Last Edit: December 5th, 2012, blt
		- Added Slave State Message Variables
	Version 20131001:
	- Added extra Output slice for motor disconnect, r.remillard


*)
TYPE udt_RobotDiscreteNode_ImageSSCCv46_20131001 :
	STRUCT
		T01: udt_EK1100;				(*Ecat Bus Coupler*)
		T02_STAT: udt_EL6900_STAT_20160426;	(*EL Safety CPU*)
		T02_CMD: udt_EL6900_CMD_20121204;
		T03: udt_EL1904_v2;				(*EL Safety Inputs*)
		T04: udt_EL1904_v2;				(*EL Safety Inputs*)
		T05: udt_EL1904_v2;				(*EL Safety Inputs*)
		T06: udt_EL1904_v2;				(*EL Safety Inputs*)
		T07: udt_EL1904_v2;				(*EL Safety Inputs*)
		T08: udt_EL2904RO_v2;			(*EL Safety Outputs, Set to "I" as this terminal is safety rated, therefore read only!*)
		T09: udt_EL2904RO_v2; 			(*EL Safety Outputs, Set to "I" as this terminal is safety rated, therefore read only!*)
		T10: udt_EL2904RO_v2; 			(*EL Safety Outputs, Set to "I" as this terminal is safety rated, therefore read only!*)
		T11: udt_EL6731;			   		(*EL Profibus Master Terminal*)
		Profinode_Stat: udt_ProfiNode_Status; 	(*Status Image of Profibus Node*)
	END_STRUCT
END_TYPE

// ---- Data types/Discrete Image udts/udt_SDx_Image.TcDUT
TYPE udt_SDx_Image :
	STRUCT
		T01: udt_EK1100;
		T02: udt_EL1904;
		T03: udt_EL2904RO;		(*Set to "I" as this terminal is safety rated, therefore read only!*)
		(*Develop Drive Nodes*)
		(*D10_STAT: udt_AX51xx_STAT;	(*Status Data Area for Drive10 (LH)*)
		D10_CMD: udt_AX51xx_CMD;		(*Command Data Area for Drive20 (RH)*)
		D20_STAT: udt_AX51xx_STAT;	(*Status Data Area for Drive10 (LH)*)
		D20_CMD: udt_AX51xx_CMD;*)		(*Command Data Area for Drive20 (RH)*)

	END_STRUCT
END_TYPE

// ---- Data types/Discrete Image udts/udt_SSxx_Image_20150814.TcDUT
(*udt (user defined type) for all generic SS (Services Stand) I/O Required
	auth. Brent Lekx-Toniolo of Sodecia GTAC

------------------------------------------------------------------------
REVISION NOTES:

	Version 20150814:
	- initial concept, b.lekx-toniolo (broken from original udt created by r.remillard)	
------------------------------------------------------------------------

*)

TYPE udt_SSxx_Image_20150814 :
STRUCT

			N01: 							udt_EP2028_002_v2;
			N01_STAT: 						udt_EP2028_002_STAT;
			N02: 							udt_EP1008_002_v2;

END_STRUCT
END_TYPE

// ---- Data types/Discrete Image udts/udt_SSxx_Image_20250704.TcDUT
(*udt (user defined type) for all generic SS (Services Stand) I/O Required
	auth. Brent Lekx-Toniolo of Sodecia GTAC

------------------------------------------------------------------------
REVISION NOTES:

	Version 20150814:
	- initial concept, b.lekx-toniolo (broken from original udt created by r.remillard)	
	Version 20250714:
	- Added in 9128, and 9214. Rearranged N02/N03, r.jones
------------------------------------------------------------------------

*)

TYPE udt_SSxx_Image_20250704 :
STRUCT
	N01: 							udt_EP9128_20250704;
	N02: 							udt_EP1008_002_v2;
	N03: 							udt_EP2028_002_v2;
	N03_STAT: 						udt_EP2028_002_STAT;
	N04_CMD: 						udt_EP9214_CMD_20250704;
	N04_STAT: 						udt_EP9214_STAT_20250704;
		
	(*Optional Power Distribution Blocks*)
	N999_STAT AT %I*: udt_EP9214_STAT_20250704;
	N999_CMD AT %Q*: udt_EP9214_CMD_20250704;
	N1000_STAT AT %I*: udt_EP9214_STAT_20250704;
	N1000_CMD AT %Q*: udt_EP9214_CMD_20250704;
	N1001_STAT AT %I*: udt_EP9214_STAT_20250704;
	N1001_CMD AT %Q*: udt_EP9214_CMD_20250704;	
	Option_EP9214_Count: INT;
			
END_STRUCT
END_TYPE

// ---- Data types/Discrete Image udts/udt_STxx_DiscreteNode_20200212.TcDUT
(*
udt (user defined type) for Visualization of Stud Weld Controller Discrete I/O Module
	Author(S): Brent Lekx-Toniolo of Sodecia GTAC;
---------------------------------------------------------------------------------------------
REVISION NOTES:

	Version 20121204
		- Intiial Concept
	Version 20200212
		- Copied from old "Nelson" named udt, abstraced name only, no code changes, b.lekx-toniolo
---------------------------------------------------------------------------------------------
*)
TYPE udt_STxx_DiscreteNode_20200212 :
	STRUCT
		T01: udt_EK1100;						(*Ecat Bus Coupler*)
		T02_STAT: udt_EL6900_STAT_20160426;	(*EL Safety CPU status*)
		T02_CMD: udt_EL6900_CMD_20121204;	(*EL Safety CPU command*)
		T03: udt_EL1904_v2;					(*EL Safety Inputs*)
		T04: udt_EL2904RO_v2;				(*EL Safety Outputs, Set to "I" as this terminal is safety rated, therefore read only!*)
		T05: udt_EL6731;						(*EL Profibus Mater Terminal*)
		Profinode_Stat: udt_ProfiNode_Status; 	(*Status Image of Profibus Node*)
	END_STRUCT
END_TYPE

// ---- Data types/Discrete Image udts/udt_WaterStand_Image_20220131.TcDUT
(*udt (user defined type) for Visualization of Water Stand Discrete I/O and Data for Visualization on UI(s)
	Author(S): Brent Lekx-Toniolo;
	Version 20151103
		- Initial Concept,blt
	Version 20200710
		- changed from EP3174 to EP6224 on N01, j.vandongen
		- removed N02 EP2028. changed to N01_CMD for EP6224, j.vandongen
	Version 20220131
		- added N01_I For UI Visualization, a.lopez


*)
TYPE udt_WaterStand_Image_20220131 :
	STRUCT

		N01: udt_EP6224;
		N01_I: udt_EP6224_I;
		N01_CMD: udt_EP6224_CMD;

		(*Cable Break States*)
		ECatSlave_Cable_Breaks: UDINT;

		(*Data developed from discrete data*)
		Water_Temp_Gun: REAL;
		Water_Temp_Trans: REAL;
		Water_Flow_Gun: REAL;
		Water_Flow_Trans: REAL;

	END_STRUCT
END_TYPE

// ---- Data types/Emhart udts/udt_Emhart_DCE1800_Inputold.TcDUT
(*udt (user defined type) of Emhart DCE 1800 Profibus Based Stud:
	auth. Brent Lekx-Toniolo of Toniolo Research & Development Inc.; 
	Sept 2010; version 1.0*)


TYPE udt_Emhart_DCE1800_Inputold :
	STRUCT
		(*Status Of Profibus Slave*)
		Inputs:udt_ProfiNode_Status;
		(*Input Bytes*)
		Byte0: USINT;
		Byte1: USINT;
		Byte2: USINT;
	END_STRUCT
END_TYPE

// ---- Data types/Emhart udts/udt_Emhart_DCE1800_Outputold.TcDUT
(*udt (user defined type) of Emhart DCE 1800 Profibus Based Stud:
	auth. Brent Lekx-Toniolo of Toniolo Research & Development Inc.; 
	Sept 2010; version 1.0*)


TYPE udt_Emhart_DCE1800_Outputold :
	STRUCT
		(*Output Bytes*)
		Byte0: USINT;
		Byte1: USINT;
		Byte2: USINT;
	END_STRUCT
END_TYPE

// ---- Data types/Emhart udts/udt_Emhart_TE1500_Input.TcDUT
(*udt (user defined type) of Emhart TE 1500 Profibus Based Stud:
	auth. Jessy Underhill; 
	Jan 2020; version 1.0*)


TYPE udt_Emhart_TE1500_Input :
	STRUCT
		(*Status Of Profibus Slave*)
		Inputs:udt_ProfiNode_Status;
		(*Input Bytes*)
		Byte0: BYTE;
		Byte1: BYTE;
		Byte2: BYTE;
		Byte3: BYTE;
		Byte4: BYTE;
		Byte5: BYTE;
		Byte6: BYTE;
		Byte7: BYTE;
	END_STRUCT
END_TYPE

// ---- Data types/Emhart udts/udt_Emhart_TE1500_Inputa.TcDUT
(*udt (user defined type) of Emhart TE 1500 Profibus Based Stud:
	auth. Jessy Underhill; 
	Jan 2020; version 1.0*)


TYPE udt_Emhart_TE1500_Inputa :
	STRUCT
		(*Status Of Profibus Slave*)
		Inputs:udt_ProfiNode_Status;
		(*Input Bytes*)
		Byte0: BYTE;
		Byte1: BYTE;
		Byte2: BYTE;
		Byte3: BYTE;
		Byte4: BYTE;
		Byte5: BYTE;
		Byte6: BYTE;
		Byte7: BYTE;
	END_STRUCT
END_TYPE

// ---- Data types/Emhart udts/udt_Emhart_TE1500_Output.TcDUT
(*udt (user defined type) of Emhart TE 1500 Profibus Based Stud:
	auth. Jessy Underhill; 
	Jan 2020; version 1.0*)


TYPE udt_Emhart_TE1500_Output :
	STRUCT
		(*Output Bytes*)
		Byte0: BYTE;
		Byte1: BYTE;
		Byte2: BYTE;
		Byte3: BYTE;
		Byte4: BYTE;
		Byte5: BYTE;
		Byte6: BYTE;
		Byte7: BYTE;
	END_STRUCT
END_TYPE

// ---- Data types/Emhart udts/udt_Emhart_TE1500_Outputa.TcDUT
(*udt (user defined type) of Emhart TE 1500 Profibus Based Stud:
	auth. Jessy Underhill; 
	Jan 2020; version 1.0*)


TYPE udt_Emhart_TE1500_Outputa :
	STRUCT
		(*Output Bytes*)
		Byte0: BYTE;
		Byte1: BYTE;
		Byte2: BYTE;
		Byte3: BYTE;
		Byte4: BYTE;
		Byte5: BYTE;
		Byte6: BYTE;
		Byte7: BYTE;
	END_STRUCT
END_TYPE

// ---- Data types/FSoE udts/ST_FSoE_02Byte.TcDUT
TYPE ST_FSoE_02Byte :
STRUCT
	CMD		: BYTE;
	SafeData1 	: WORD;
	CRC1		: WORD;
	ConnID		: WORD;
END_STRUCT
END_TYPE

// ---- Data types/FSoE udts/ST_FSoE_04Byte.TcDUT
TYPE ST_FSoE_04Byte :
STRUCT
	CMD		: BYTE;
	SafeData1 	: WORD;
	CRC1		: WORD;
	SafeData2 	: WORD;
	CRC2		: WORD;
	ConnID		: WORD;
END_STRUCT
END_TYPE

// ---- Data types/FSoE udts/ST_FSoE_06Byte.TcDUT
TYPE ST_FSoE_06Byte :
STRUCT
	CMD		: BYTE;
	SafeData1 	: WORD;
	CRC1		: WORD;
	SafeData2 	: WORD;
	CRC2		: WORD;
	SafeData3 	: WORD;
	CRC3		: WORD;
	ConnID		: WORD;
END_STRUCT
END_TYPE

// ---- Data types/FSoE udts/ST_FSoE_08Byte.TcDUT
TYPE ST_FSoE_08Byte :
STRUCT
	CMD		: BYTE;
	SafeData1 	: WORD;
	CRC1		: WORD;
	SafeData2 	: WORD;
	CRC2		: WORD;
	SafeData3 	: WORD;
	CRC3		: WORD;
	SafeData4 	: WORD;
	CRC4		: WORD;
	ConnID		: WORD;
END_STRUCT
END_TYPE

// ---- Data types/FSoE udts/ST_FSoE_10Byte.TcDUT
TYPE ST_FSoE_10Byte :
STRUCT
	CMD		: BYTE;
	SafeData1 	: WORD;
	CRC1		: WORD;
	SafeData2 	: WORD;
	CRC2		: WORD;
	SafeData3 	: WORD;
	CRC3		: WORD;
	SafeData4 	: WORD;
	CRC4		: WORD;
	SafeData5 	: WORD;
	CRC5		: WORD;
	ConnID		: WORD;
END_STRUCT
END_TYPE

// ---- Data types/FSoE udts/ST_FSoE_12Byte.TcDUT
TYPE ST_FSoE_12Byte :
STRUCT
	CMD		: BYTE;
	SafeData1 	: WORD;
	CRC1		: WORD;
	SafeData2 	: WORD;
	CRC2		: WORD;
	SafeData3 	: WORD;
	CRC3		: WORD;
	SafeData4 	: WORD;
	CRC4		: WORD;
	SafeData5 	: WORD;
	CRC5		: WORD;
	SafeData6 	: WORD;
	CRC6		: WORD;
	ConnID		: WORD;
END_STRUCT
END_TYPE

// ---- Data types/FSoE udts/ST_FSoE_14Byte.TcDUT
TYPE ST_FSoE_14Byte :
STRUCT
	CMD		: BYTE;
	SafeData1 	: WORD;
	CRC1		: WORD;
	SafeData2 	: WORD;
	CRC2		: WORD;
	SafeData3 	: WORD;
	CRC3		: WORD;
	SafeData4 	: WORD;
	CRC4		: WORD;
	SafeData5 	: WORD;
	CRC5		: WORD;
	SafeData6 	: WORD;
	CRC6		: WORD;
	SafeData7 	: WORD;
	CRC7		: WORD;
	ConnID		: WORD;
END_STRUCT
END_TYPE

// ---- Data types/Generic udts/udt_Generic_AdsAddr.TcDUT
(*udt (user defined type) of Beckhoff EK1100 - EtherCAT Bus Coupler (Slave):
	auth. Brent Lekx-Toniolo of Toniolo Research & Development Inc.; 
	July 2010; version 1.0*)


TYPE udt_Generic_AdsAddr :
	STRUCT
		netId: ARRAY[0..5] OF USINT;
		port: UINT;
	END_STRUCT
END_TYPE

// ---- Data types/Generic udts/udt_Generic_EP9214_20250714.TcDUT
TYPE udt_Generic_EP9214_20250714 :
STRUCT		

	Safety_RST: BOOL;
	Enable_Motion: BOOL;
	Prev_EcatNode_Present: BOOL;
	Option_EP9214_Count: INT;
	
	Channel1_Output_Us: BOOL;
	Channel1_Output_Up: BOOL;
	Channel1_Reset_Us: BOOL;
	Channel1_Reset_Up: BOOL;
	
	Channel2_Output_Us: BOOL;
	Channel2_Output_Up: BOOL;
	Channel2_Reset_Us: BOOL;
	Channel2_Reset_Up: BOOL;
	
	Channel3_Output_Us: BOOL;
	Channel3_Output_Up: BOOL;
	Channel3_Reset_Us: BOOL;
	Channel3_Reset_Up: BOOL;
	
	Channel4_Output_Us: BOOL;
	Channel4_Output_Up: BOOL;
	Channel4_Reset_Us: BOOL;
	Channel4_Reset_Up: BOOL;
	
	
END_STRUCT
END_TYPE

// ---- Data types/Generic udts/udt_Generic_IC_20150928.TcDUT
(*
udt (user defined type) for all generic IC (Industrical Controller Panel) Data Required
	auth. Brent Lekx-Toniolo of Toniolo Research & Development Inc.; 
	August 2010; version 1.0

	Version 20150120:
	- Updated name to include date rev, b.lekx-toniolo
	- Added "previous ecat node present" input, b.lekx-toniolo
	Version 20150928:
	- Added Ecat_Master_AmsNetID, CoE_Read_Trigger, b.lekx-toniolo

*)
TYPE udt_Generic_IC_20150928 :
	STRUCT
		Safety_RST: BOOL;
		Enable_Motion: BOOL;
		Estops_OK: BOOL;
		Safety_Gates_Ok: BOOL;
		Ecat_Master_AmsNetID: STRING;
		CoE_Read_Trigger: BOOL;
		Prev_EcatNode_Present: BOOL;
		OP1_Green_LampReq: BOOL;
		OP1_Yellow_LampReq: BOOL;
		OP1_Red_LampReq: BOOL;
		OP1_Audible_Req: BOOL;
		OP2_Green_LampReq: BOOL;
		OP2_Yellow_LampReq: BOOL;
		OP2_Red_LampReq: BOOL;
		OP2_Audible_Req: BOOL;
		Output_Req1: BOOL;
		Output_Req2: BOOL;


	END_STRUCT
END_TYPE

// ---- Data types/Generic udts/udt_Generic_Nok_Data_Grid_20251208.TcDUT
TYPE udt_Generic_Nok_Data_Grid_20251208 :
STRUCT
	TimeStamp : STRING;
	Model_ID : STRING;
	NOK_Faulted : STRING;    
	Unload_Completed : BOOL; (*reset signal*)
	
END_STRUCT
END_TYPE

// ---- Data types/Generic udts/udt_Generic_NutWeldLVDTConfig_20250612.TcDUT
(*udt (user defined type) for nut weld LVDT config data (developed from some code in project 21013_1

	Author(S): Brent Lekx-Toniolo ;
	Version 20250612:
		- Initial Concept

*)



TYPE udt_Generic_NutWeldLVDTConfig_20250612 :
STRUCT
	
	Pin_ADVD_UpperLimit: REAL;		(*Upper limit for the Pin ADVD Range*)
	Pin_ADVD_LowerLimit: REAL;		(*Lower limit for the Pin ADVD Range*)
	Pin_RETD_UpperLimit: REAL;		(*Upper limit for the Pin RETD Range*)
	Pin_RETD_LowerLimit: REAL;		(*Lower limit for the Pin RETD Range*)
	Nut_UpperLimit: REAL;			(*Upper limit for the Nut present range on Pin*)
	Nut_LowerLimit: REAL;			(*Lower limit for the Nut present range on Pin*)
	UpperElectrode_WeldCountLimit: UINT;	(*Weld Count limit for System Upper Electrode (for wear)*)
END_STRUCT
END_TYPE

// ---- Data types/Generic udts/udt_Generic_PD_20220906.TcDUT
(*udt (user defined type) for all generic PD (Power Distribution Panel) Data Required
	auth. Brent Lekx-Toniolo of Toniolo Research & Development Inc.; 
	August 2010; version 1.0

	Version 20150812:
	- Updated name to include date rev, b.lekx-toniolo
	- Modified per V5.00 requirements, b.lekx-toniolo
	Version 20150928:
	- Added Ecat_Master_AmsNetID, CoE_Read_Trigger, b.lekx-toniolo
	Version 20170307
	- Added Enable Inputs for Split Relays and EP9224, b.lekx-toniolo
	Version 20190924
	- added Enable to Profibus (EL6731), j.vandongen
	Version 20220906
	-Changed Boolean Enable to numerical Count for EP9224 , C.Drees


*)

TYPE udt_Generic_PD_20220906:
	STRUCT
		Safety_RST: BOOL;
		Enable_Motion: BOOL;
		Ecat_Master_AmsNetID: STRING;
		CoE_Read_Trigger: BOOL;
		Prev_EcatNode_Present: BOOL;
		Option_Enable_SplitRelays: BOOL;
		Option_EP9224_Count: INT;
		Option_Enable_Pbus: BOOL;

	END_STRUCT
END_TYPE

// ---- Data types/Generic udts/udt_Generic_Production_20221007.TcDUT
(*udt (user defined type) for production report data

	Author(S): Rob Remillard and Brent Lekx-Toniolo ;
	V1:
		- Initial Concept
	
	Version 20160229:
		- Increase Expected_Count Array size from 8 to 12, b.lekx-toniolo
		- Enabled Start and End of Shift Time Structs, b.lekx-toniolo
		- Added Report Status String, b.lekx-toniolo
		- Changed PPH to REAL, b.lekx-toniolo
	Version 20191125:
		- Added fault count, running up time and net shift duration time, b.lekx-toniolo
	Version 20221007:
		- Added in Target CT to capture this value within the report itself, b.lekx-toniolo	
*)


TYPE udt_Generic_Production_20221007 :
	STRUCT
	(*----------- Data Area For Tagging Report with Machine Name, Date and Operator ID ----------*)
	Machine_Serial: STRING;
	Machine_Common_Name: STRING;
	(*Logged in Operator ID*)
	Operator_ID: UINT;
	(*Data Area For Tagging Report with Shift Times and Date*)
	Start_Shift_TimeDate: TIMEStruct;
	End_Shift_TimeDate: TIMEStruct;
	(*Target Cycle Time*)
	Target_Cycle_Time: TIME;

	(*------------ Shift Configuration --------------*)

	ProdConfig_Common: udt_Generic_ShiftCommonConfig_20220420;
	ProdConfig_Times: udt_Generic_ShiftConfigUDINT_20160531;

	(*---------------- Hourly Report ---------------*)
	(*Running Total Production Count After Each Hour*)
	Total_Count: ARRAY[0..12] OF UINT;
	(*Total Production Count OF Each Hour*)
	Hour_Count: ARRAY[0..12] OF UINT;
	(*Hourly Expected Count*)
	Expected_Count: ARRAY[0..12] OF UINT;
	(*Final Production Total Including Scrap, GROSS Production*)
	Prod_Count_Total: UINT;
	(*Total Scrap Made During Shift*)
	Prod_Count_Scrap:UINT;

	(*------------- OEE KPI Metrics ---------------*)

	(*Availability*)
	Prod_Availability: REAL;
	(*Running Performance*)
	Prod_Performance: REAL;
	(*Running Quality*)
	Prod_Quality: REAL;
	(*Running OEE*)
	Prod_Running_OEE: REAL;

	(*----------- Misc Numbers -----------------*)
	(*Static Production Target*)
	Prod_Static_Target: UINT;
	(*Incrementing Target (Tac Time)*)
	Prod_Running_Target: UINT;
	(*Calced Difference Of Above*)
	Prod_Difference: DINT;
	(*Final Average PPH*)
	Prod_AvgFinal_PPH: REAL;
	(*Total Machine Fault Time*)
	Total_Fault_Time: TIME;
	(*Fault Count During Shift*)
	Total_Fault_Count: UDINT;
	(*Running Up Time*)
	Running_Up_Time: TIME;
	(*Shift Durations, Gross = End time - Start Time, Net = Gross -  breaks and optional expected downtime*)
	Gross_Shift_Duration: REAL;
	Net_Shift_Duration: REAL;

	(*--------------- Report Status --------------*)
	Status: STRING;



	END_STRUCT
END_TYPE

// ---- Data types/Generic udts/udt_Generic_ProductReportData_20240909.TcDUT
(*udt (user defined type) for product report data 
Product report data can be populated with part / assembly / product measurements etc etc

	Author(S): Version 20221007:
		- Initial concept, b.lekx-toniolo and c.drees during tcui migration	
	Version 20240909:
		- Added in Model_Id and Spare Areas, b.lekx-toniolo
*)



TYPE udt_Generic_ProductReportData_20240909 :
STRUCT
	
	(*Machine Indentifiers*)
	Machine_Serial: STRING;
	Machine_Common_Name: STRING;
	(*Operator Identifier*)
	Operator_ID: UINT;
	(*Product Identifier*)
	Product_Serial: STRING; 
	Product_Number: STRING;
	Product_Common_Name: STRING;
	Product_Model_ID: UINT;
	(*Spare Areas for general use*)
	Spare1: STRING;
	Spare2: STRING;
	
	(*Generic pass fail array*)
	Generic_PassFail_Notes: ARRAY[0..31] OF STRING(4);
	
	(*Generic measurement array*)
	Generic_Measurements: ARRAY [0..31] OF REAL;
	
END_STRUCT
END_TYPE

// ---- Data types/Generic udts/udt_Generic_Robot_20161202.TcDUT
(*udt (user defined type) for all generic Robot Data Required
	Author(S): Brent Lekx-Toniolo of Sodecia GTAC;
	Version 1.0: August 2010
		- Initial Concept
	Version 2.0: November 2012
		- Expanded Equipment Interf Area
		- Expanded Elements in each Array for more inter zone data areas
	Version 20141014
		- added RobotInters, b.lekx-toniolo
	Version 20161202
		- added AuxReq_Aux, j.vandongen

*)



TYPE udt_Generic_Robot_20161202 :
	STRUCT
		Safety_RST: BOOL;
		Enable_Motion: BOOL;
		Alarm_RST: BOOL;
		Robot_Type: UINT;
		Select_Play: BOOL;
		Select_Teach: BOOL;
		Select_Remote: BOOL;
		Start_Scan: BOOL;
		Stop_Scan: BOOL;
		Stop_Scan2: BOOL;
		In_DryCycle: BOOL;
		Low_Speed: BOOL;
		Major_Faults: BOOL;
		Teach_Interlock: BOOL;
		Weld_Inhibit: BOOL;
		Power_Disable: BOOL;

		OK_ToEnter_EquipInterf1: BOOL;
		OK_ToEnter_EquipInterf2: BOOL;
		OK_ToEnter_EquipInterf3: BOOL;
		OK_ToEnter_EquipInterf4:  BOOL;
		OK_ToEnter_EquipInterf5: BOOL;
		OK_ToEnter_EquipInterf6: BOOL;
		OK_ToEnter_EquipInterf7: BOOL;
		OK_ToEnter_EquipInterf8:  BOOL;
		OK_ToEnter_EquipInterf9:  BOOL;
		OK_ToEnter_HumanInterf1: BOOL;
		OK_ToEnter_HumanInterf2: BOOL;
		OK_ToEnter_HumanInterf3: BOOL;
		OK_ToEnter_HumanInterf4: BOOL;
		OK_ToEnter_HumanInterf5: BOOL;
		OK_ToEnter_HumanInterf6: BOOL;
		OK_ToEnter_HumanInterf7: BOOL;
		OK_ToEnter_HumanInterf8: BOOL;

		OK_ToEnter_RobotInterfs: UINT;

		Fix_ID: ARRAY [0..17] OF UINT;
		EOAT_ID: ARRAY [0..17] OF UINT;
		Model_ID: ARRAY [0..17] OF  UINT;
		Task_ID: ARRAY [0..17] OF UINT;
		PeripheralReq_Ack: ARRAY [0..17] OF UINT;
		AuxReq_Ack: ARRAY [0..17] OF UINT;

		Proceed_From_Pounce: ARRAY[0..17] OF BOOL;
		Complete_Ack: ARRAY[0..17] OF BOOL;

	END_STRUCT
END_TYPE

// ---- Data types/Generic udts/udt_Generic_Robot_20250711_CUSTOM.TcDUT
(*udt (user defined type) for all generic Robot Data Required
	Author(S): Brent Lekx-Toniolo of Sodecia GTAC;
	Version 1.0: August 2010
		- Initial Concept
	Version 2.0: November 2012
		- Expanded Equipment Interf Area
		- Expanded Elements in each Array for more inter zone data areas
	Version 20141014
		- added RobotInters, b.lekx-toniolo
	Version 20161202
		- added AuxReq_Aux, j.vandongen
	Version 20250711_CUSTOM
		- added OK_ToEnter_EquipInterf9, w.griffiths

*)



TYPE udt_Generic_Robot_20250711_CUSTOM :
	STRUCT
		Safety_RST: BOOL;
		Enable_Motion: BOOL;
		Alarm_RST: BOOL;
		Robot_Type: UINT;
		Select_Play: BOOL;
		Select_Teach: BOOL;
		Select_Remote: BOOL;
		Start_Scan: BOOL;
		Stop_Scan: BOOL;
		Stop_Scan2: BOOL;
		In_DryCycle: BOOL;
		Low_Speed: BOOL;
		Major_Faults: BOOL;
		Teach_Interlock: BOOL;
		Weld_Inhibit: BOOL;
		Power_Disable: BOOL;

		OK_ToEnter_EquipInterf1: BOOL;
		OK_ToEnter_EquipInterf2: BOOL;
		OK_ToEnter_EquipInterf3: BOOL;
		OK_ToEnter_EquipInterf4:  BOOL;
		OK_ToEnter_EquipInterf5: BOOL;
		OK_ToEnter_EquipInterf6: BOOL;
		OK_ToEnter_EquipInterf7: BOOL;
		OK_ToEnter_EquipInterf8:  BOOL;
		OK_ToEnter_EquipInterf9:  BOOL;
		OK_ToEnter_HumanInterf1: BOOL;
		OK_ToEnter_HumanInterf2: BOOL;
		OK_ToEnter_HumanInterf3: BOOL;
		OK_ToEnter_HumanInterf4: BOOL;
		OK_ToEnter_HumanInterf5: BOOL;
		OK_ToEnter_HumanInterf6: BOOL;
		OK_ToEnter_HumanInterf7: BOOL;
		OK_ToEnter_HumanInterf8: BOOL;

		OK_ToEnter_RobotInterfs: UINT;

		Fix_ID: ARRAY [0..17] OF UINT;
		EOAT_ID: ARRAY [0..17] OF UINT;
		Model_ID: ARRAY [0..17] OF  UINT;
		Task_ID: ARRAY [0..17] OF UINT;
		PeripheralReq_Ack: ARRAY [0..17] OF UINT;
		AuxReq_Ack: ARRAY [0..17] OF UINT;

		Proceed_From_Pounce: ARRAY[0..17] OF BOOL;
		Complete_Ack: ARRAY[0..17] OF BOOL;

	END_STRUCT
END_TYPE

// ---- Data types/Generic udts/udt_Generic_Robot_FBIN_CUSTOM.TcDUT
(*udt (user defined type) for all generic Robot Data Required
	Author(S): Brent Lekx-Toniolo of Sodecia GTAC;
	Version 1.0: August 2012
		- Initial Concept
	 Version 2.0: November 2012,
		Changes from v1 include:
			- Expanded Equipment Interf Area
			- Added EOAT Req Ack
			-Added Water_OK Inputs (to be sent to WCUs)
			- Added Water Output Command Bit (For Control of Slaves via Robot)
			- Added EOAT Output Command Areas (For Control of Slaves via Robot)
	Version: 20130625
			- Added Speed Request Var
	Version 20141016:
			- Added WeldCont_Amount, to give ability to select amount of weld controllers robot will interface to, b.lekx-toniolo
			- Added Under_Construction Input to remove external dependancy on variable, b.lekx-toniolo
			- Added OK to enter Robot Infer Inputs to break away from equip interf area, b.lekx-toniolo
			- Added Install_Zero_Orientation for use with new UI Robot Animation Symbol, b.lekx-toniolo
	Version 20150103:
			- Added SOS_Requested. RR/JVD
	Version 20150120:
			- Added "previous ecat node present" input, b.lekx-toniolo
	Version 20150318:
			- Added "Force Master and Brake Test Reqs", b.lekx-toniolo
	Version 20150928:
			- Added Ecat_Master_AmsNetID, CoE_Read_Trigger, b.lekx-toniolo
	Version 20160127:
			- Removed old Water Interface and Added config interface, part of internalizing water stand code, b.lekx-toniolo
	Version 20160203:
			- Added Option Enable Variables, b.lekx-toniolo
	Version 20161202:
			-added Aux Request ACK, j.vandongen
	Version 20170531:
			- Updated instance of Options, b.lekx-toniolo
	Version 20170801:
			- updated instance of options, j.vandongen
	Version 20190923
			- added EOAT_FLT variable, j.vandongen
	Version 20240208
			- added In_Sim_Mode and SIM_StartWorkAround during R&D project 90034, sim integration, b.lekx-toniolo
			- Correct some minor typos etc to do with Disable water fault (FB Input), b.lekx-toniolo
			

*)
TYPE udt_Generic_Robot_FBIN_CUSTOM :
	STRUCT
		Safety_RST: BOOL;
		Enable_Motion: BOOL;
		Alarm_RST: BOOL;
		Robot_Type: UINT;
		Install_Zero_Orientation: INT;
		Under_Construction: BOOL;
		In_SIM_Mode: BOOL;
		SIM_StartWorkAround: BOOL;
		
		Ecat_Master_AmsNetID: STRING;
		CoE_Read_Trigger: BOOL;
		Prev_EcatNode_Present: BOOL;
		Select_Play: BOOL;
		Select_Teach: BOOL;
		Select_Remote: BOOL;
		Start_Scan: BOOL;
		Stop_Scan: BOOL;
		Stop_Scan2: BOOL;
		In_DryCycle: BOOL;
		Low_Speed: BOOL;
		Major_Faults: BOOL;
		Teach_Interlock: BOOL;
		Weld_Inhibit: BOOL;
		Power_Disable: BOOL;
		Force_MasterTest_Req: BOOL;
		Force_BrakeTest_Req: BOOL;
		EOAT_FLT: BOOL;

		Speed_Request: BYTE;
		OK_ToEnter_EquipInterf1: BOOL;
		OK_ToEnter_EquipInterf2: BOOL;
		OK_ToEnter_EquipInterf3: BOOL;
		OK_ToEnter_EquipInterf4: BOOL;
		OK_ToEnter_EquipInterf5: BOOL;
		OK_ToEnter_EquipInterf6: BOOL;
		OK_ToEnter_EquipInterf7: BOOL;
		OK_ToEnter_EquipInterf8: BOOL;
		OK_ToEnter_EquipInterf9: BOOL;
		OK_ToEnter_HumanInterf1: BOOL;
		OK_ToEnter_HumanInterf2: BOOL;
		OK_ToEnter_HumanInterf3: BOOL;
		OK_ToEnter_HumanInterf4: BOOL;
		OK_ToEnter_HumanInterf5: BOOL;
		OK_ToEnter_HumanInterf6: BOOL;
		OK_ToEnter_HumanInterf7: BOOL;
		OK_ToEnter_HumanInterf8: BOOL;

		OK_ToEnter_RobotInterfs: UINT;

		User_Inputs: BYTE;

		Fix_ID: UINT;
		Task_ID: UINT;
		Model_ID: UINT;
		EOAT_ID: UDINT;
		PeripheralReq_Ack: UINT;
		AuxReq_Ack: UINT;
		EOATReq_Ack: UINT;

		Proceed_From_Pounce: BOOL;
		Complete_Ack: BOOL;

		Option_Disable_WaterFLT: BOOL;	

		SOS_Requested: BOOL;

		(*Option Configuration Inputs*)
		Options: udt_Generic_Robot_Options_20170531;

	END_STRUCT
END_TYPE

// ---- Data types/Generic udts/udt_Generic_Robot_FBIN_20250711_CUSTOM.TcDUT
(*udt (user defined type) for all generic Robot Data Required
	Author(S): Brent Lekx-Toniolo of Sodecia GTAC;
	Version 1.0: August 2012
		- Initial Concept
	 Version 2.0: November 2012,
		Changes from v1 include:
			- Expanded Equipment Interf Area
			- Added EOAT Req Ack
			-Added Water_OK Inputs (to be sent to WCUs)
			- Added Water Output Command Bit (For Control of Slaves via Robot)
			- Added EOAT Output Command Areas (For Control of Slaves via Robot)
	Version: 20130625
			- Added Speed Request Var
	Version 20141016:
			- Added WeldCont_Amount, to give ability to select amount of weld controllers robot will interface to, b.lekx-toniolo
			- Added Under_Construction Input to remove external dependancy on variable, b.lekx-toniolo
			- Added OK to enter Robot Infer Inputs to break away from equip interf area, b.lekx-toniolo
			- Added Install_Zero_Orientation for use with new UI Robot Animation Symbol, b.lekx-toniolo
	Version 20150103:
			- Added SOS_Requested. RR/JVD
	Version 20150120:
			- Added "previous ecat node present" input, b.lekx-toniolo
	Version 20150318:
			- Added "Force Master and Brake Test Reqs", b.lekx-toniolo
	Version 20150928:
			- Added Ecat_Master_AmsNetID, CoE_Read_Trigger, b.lekx-toniolo
	Version 20160127:
			- Removed old Water Interface and Added config interface, part of internalizing water stand code, b.lekx-toniolo
	Version 20160203:
			- Added Option Enable Variables, b.lekx-toniolo
	Version 20161202:
			-added Aux Request ACK, j.vandongen
	Version 20170531:
			- Updated instance of Options, b.lekx-toniolo
	Version 20170801:
			- updated instance of options, j.vandongen
	Version 20190923
			- added EOAT_FLT variable, j.vandongen
	Version 20240208
			- added In_Sim_Mode and SIM_StartWorkAround during R&D project 90034, sim integration, b.lekx-toniolo
			- Correct some minor typos etc to do with Disable water fault (FB Input), b.lekx-toniolo
	Version 20250711_CUSTOM
			- Added EquipInterf9, w.griffiths
			

*)
TYPE udt_Generic_Robot_FBIN_20250711_CUSTOM :
	STRUCT
		Safety_RST: BOOL;
		Enable_Motion: BOOL;
		Alarm_RST: BOOL;
		Robot_Type: UINT;
		Install_Zero_Orientation: INT;
		Under_Construction: BOOL;
		In_SIM_Mode: BOOL;
		SIM_StartWorkAround: BOOL;
		
		Ecat_Master_AmsNetID: STRING;
		CoE_Read_Trigger: BOOL;
		Prev_EcatNode_Present: BOOL;
		Select_Play: BOOL;
		Select_Teach: BOOL;
		Select_Remote: BOOL;
		Start_Scan: BOOL;
		Stop_Scan: BOOL;
		Stop_Scan2: BOOL;
		In_DryCycle: BOOL;
		Low_Speed: BOOL;
		Major_Faults: BOOL;
		Teach_Interlock: BOOL;
		Weld_Inhibit: BOOL;
		Power_Disable: BOOL;
		Force_MasterTest_Req: BOOL;
		Force_BrakeTest_Req: BOOL;
		EOAT_FLT: BOOL;

		Speed_Request: BYTE;
		OK_ToEnter_EquipInterf1: BOOL;
		OK_ToEnter_EquipInterf2: BOOL;
		OK_ToEnter_EquipInterf3: BOOL;
		OK_ToEnter_EquipInterf4: BOOL;
		OK_ToEnter_EquipInterf5: BOOL;
		OK_ToEnter_EquipInterf6: BOOL;
		OK_ToEnter_EquipInterf7: BOOL;
		OK_ToEnter_EquipInterf8: BOOL;
		OK_ToEnter_EquipInterf9: BOOL;
		OK_ToEnter_HumanInterf1: BOOL;
		OK_ToEnter_HumanInterf2: BOOL;
		OK_ToEnter_HumanInterf3: BOOL;
		OK_ToEnter_HumanInterf4: BOOL;
		OK_ToEnter_HumanInterf5: BOOL;
		OK_ToEnter_HumanInterf6: BOOL;
		OK_ToEnter_HumanInterf7: BOOL;
		OK_ToEnter_HumanInterf8: BOOL;

		OK_ToEnter_RobotInterfs: UINT;

		User_Inputs: BYTE;

		Fix_ID: UINT;
		Task_ID: UINT;
		Model_ID: UINT;
		EOAT_ID: UDINT;
		PeripheralReq_Ack: UINT;
		AuxReq_Ack: UINT;
		EOATReq_Ack: UINT;

		Proceed_From_Pounce: BOOL;
		Complete_Ack: BOOL;

		Option_Disable_WaterFLT: BOOL;

		SOS_Requested: BOOL;

		(*Option Configuration Inputs*)
		Options: udt_Generic_Robot_Options_20170531;

	END_STRUCT
END_TYPE

// ---- Data types/Generic udts/udt_Generic_Robot_Options_20170531.TcDUT
(*udt (user defined type) for generic Robot Add-In Option Configuration
	Version 20160204:
	- Initial Concept, b.lekx-toniolo
	Version 20170531:
	- Added Mig controller amount, b.lekx-toniolo


*)
TYPE udt_Generic_Robot_Options_20170531 :
	STRUCT
		(*Option Config Inputs*)
		WeldCont_Amount: UINT;
		MIGCont_Amount: UINT;
		WaterStand_Amount: UINT;
		Reamer_Amount: UINT;
		EOAT_Amount: UINT;
	END_STRUCT
END_TYPE

// ---- Data types/Generic udts/udt_Generic_Sensor_States_20170801.TcDUT
TYPE udt_Generic_Sensor_States_20170801 :
	(
	LoadOK1:=0,
	LoadOK2:=1,
	LoadOK:=2,

	StartWeld:=5,
	StartTurn:=6,
	StartSeal:=7,
	StartStud:=8,
	StartUnload1:=9,
	StartUnload2:=10,


	(*Sensor_At_Repo Positions*)
	SenseRepo0:=15,
	SenseRepo1:=16,
	SenseRepo2:=17,
	SenseRepo3:=18,
	SenseRepo4:=19,
	SenseRepo5:=20,
	SenseRepo6:=21,
	SenseRepo7:=22,
	SenseRepo8:=23,
	SenseRepo9:=24,
	SenseRepo10:=25,
	SenseRepo11:=26,
	SenseRepo12:=27,
	SenseRepo13:=28,
	SenseRepo14:=29,
	SenseRepo15:=30,
	SenseRepo16:=31

	);
END_TYPE

// ---- Data types/Generic udts/udt_Generic_ServoDrive_FBIN_20211214.TcDUT
(*
udt (user defined type) for generic FB Inputs required for GTAC standard Servo Drive Profile
	auth. Brent Lekx-Toniolo of Sodecia GTAC. 

	Version 20160809:
	- Intial concept, b.lekx-toniolo
	Version 20161124
	- Broke out sperated Enable Motions per axis
	Version 20161214
	- Added Soft Limits, b.lekx-toniolo
	- Added Home Position Inputs, b.lekx-toniolo
	- Added Direct Home Input, b.lekx-toniolo
	- Added Homing Type Input, b.lekx-toniolo
	- Added Axis_ID Input, b.lekx-toniolo
	Version 20180731
	- Added position variable to the UDT - b.donnell
	- Added teach enabled bit - b.donnell
	- Added safe tool position bit for manual mode, b.donnell
	Version 20210203
	- Added Max_Torque Inputs
	Version 20211115
	- Changed Array size from [1..15] to [0..15] for Position, and AutoControls - C.drees
	Version 20211214
	- Updates to allow input of Reference Position from outside of FB, c.drees / b.lekx-toniolo
	- Changed data types of Max_Torque vars for use to map to PDO inputs, c.drees / b.lekx-toniolo
	
*)
TYPE udt_Generic_ServoDrive_FBIN_20211214 :
STRUCT
		Enable_Motion: ARRAY[1..2] OF BOOL;
		Option_Type: UINT; 			(*0=AX5000 drive, 10=EL72xx terminal drive*)
		Option_Axis_Count: UINT;		(*Option Axis Count->  max 1 for 72xx drive, max 2 for AX52xx series drive*)
		ECAT_AmsID: STRING;
		Prev_EcatNode_Present: BOOL;

		Axis_Common_Name: ARRAY[1..2] OF STRING [30];
		Rotary_Axis: ARRAY[1..2] OF BOOL;						(*Axis is a rotary table*)
		Axis_Is_Absolute: ARRAY[1..2] OF BOOL;					(*Axis is Absolute Type*)
		System_Max_Velocity: ARRAY[1..2] OF REAL;				(*Pass Servo System Maximum Velocity in Here*)
		System_Stop_Decel: ARRAY [1..2] OF REAL;				(*Set System MC_Stop Decel rate, default hard coded in FB if not entered*)
		Soft_Limit_Max: ARRAY[1..2] OF REAL;					(*Pass Softwarer limits here*)
		Soft_Limit_Min: ARRAY[1..2] OF REAL;
		Disable_Soft_Limits: ARRAY[1..2] OF BOOL;				(*Run Servo System without Soft Limits*)
		Home_Position_Switch: ARRAY[1..2] OF BOOL;			(*Home (Callibration) switch*)
		Quick_Home_REQ: ARRAY[1..2] OF BOOL;				(*Request a quick Home where the homing request is sent to system with no delay, good for on the fly homing*)
		Homing_Type: ARRAY[1..2] OF MC_HomingMode;			(*Pass Homing Type, see beckhoff documents for various homing routine types*)
		Homing_Offset: ARRAY[1..2] OF REAL;					(*Pass Homing Offset for QuickHome*)
		MicroInch_Value: ARRAY[1..2] OF REAL;					(*Value to Micro Inch*)
		Mode_Select: ARRAY[1..2] OF INT;
		Error_Reset: ARRAY[1..2] OF BOOL;
		Program_Reset: ARRAY[1..2] OF BOOL;

		Position: ARRAY[1..2] OF ARRAY[0..15] OF REAL;
		Auto_Vel: ARRAY[1..2] OF ARRAY[0..15] OF REAL;
		Auto_Accel: ARRAY[1..2] OF ARRAY[0..15] OF REAL;
		Auto_Decel: ARRAY[1..2] OF ARRAY[0..15] OF REAL;
		Auto_MoveType: ARRAY[1..2] OF ARRAY[0..15] OF INT;
		Auto_EndFlag: ARRAY[1..2] OF ARRAY[0..15] OF BOOL;
		Teach_Enable: ARRAY[1..2] OF BOOL;
		Max_Torque: ARRAY[1..2] OF INT;
		
		PlayBack_Speed_Percentage: ARRAY[1..2] OF REAL;
		Explicit_Step_REQ: ARRAY[1..2] OF UINT;
		Start_Explicit_StepCall: ARRAY[1..2] OF BOOL;
		Start_PlayBack: ARRAY[1..2] OF BOOL;
		Stop_PlayBack: ARRAY[1..2] OF BOOL;
		PlayBack_StepPermit: ARRAY[1..2] OF BOOL;


		Safe_Tool_Pos: ARRAY[1..2] OF BOOL;
		Teach_Params: ARRAY[1..2] OF udt_SingleAxis_MoveData_20160908; (*Struct of Teach paramaeters*)
		Teach_Servo_HomePos: ARRAY[1..2] OF BOOL;
		Teach_JogFast_Plus: ARRAY[1..2] OF BOOL;
		Teach_JogFast_Minus: ARRAY[1..2] OF BOOL;
		Teach_JogSlow_Plus: ARRAY[1..2] OF BOOL;
		Teach_JogSlow_Minus: ARRAY[1..2] OF BOOL;
		Teach_Inch_Plus: ARRAY[1..2] OF BOOL;
		Teach_Inch_Minus: ARRAY[1..2] OF BOOL;
		Teach_MicroInch_Enable: ARRAY[1..2] OF BOOL;
		Teach_Record_CurrentPos: ARRAY[1..2] OF BOOL;
		Teach_ParamsOverwrite_Flag: ARRAY[1..2] OF BOOL;

END_STRUCT
END_TYPE

// ---- Data types/Generic udts/udt_Generic_ShiftCommonConfig_20220420.TcDUT
(*udt (user defined type) for production shift config common data (production config data common to all shifts)


	Author(S): Brent Lekx-Toniolo ;
	20191125:
	- Initial Concept
	2020020
	- Added a variable for Return to Defaults - C.Drees
	


*)


TYPE udt_Generic_ShiftCommonConfig_20220420 :
	STRUCT
		Config_Source: UINT;			(*Selects source data for Production Shift Configuration (current allows UI or default configs, future addition shall allow config via spreadsheet*)
		Shift_Enables: UINT;			(*Enable Flags for shifts in a 24 hour period*)
		Break_Count: UINT;			(*Amount of breaks per shift*)
		ResetProdConfig_To_Default:BOOL;
		Config_Option_Flags: UINT;
				(*
				Flags shall be used to allow bit wise configuration to the production FB	
				Current Option Flag Assignment:
					Config_Option_Flags.0 = In Shift Change Time (used to feed Enable_InShift_Change input on FB_Production_Report_yyymmdd)
					Config_Option_Flags.1 = spare
					Config_Option_Flags.2 = spare
					Config_Option_Flags.3 = spare
					Config_Option_Flags.4 = spare
					Config_Option_Flags.5 = spare
					Config_Option_Flags.6 = spare
					Config_Option_Flags.7 = spare
					Config_Option_Flags.8 = spare
					Config_Option_Flags.9 = spare
					Config_Option_Flags.10 = Save Report as file type flag (0 = xls, 1= csv)
					Config_Option_Flags.11 = spare
					Config_Option_Flags.12 = spare
					Config_Option_Flags.13 = spare
					Config_Option_Flags.14 = spare
					Config_Option_Flags.15 = spare
				*)


	END_STRUCT
END_TYPE

// ---- Data types/Generic udts/udt_Generic_ShiftConfigTOD_20160527.TcDUT
(*udt (user defined type) for production shift config data In TOD (Time Of Day) Format

	Author(S): Brent Lekx-Toniolo ;
	20160527:
		- Initial Concept
	


*)


TYPE udt_Generic_ShiftConfigTOD_20160527 :
	STRUCT
		Shift_StartTime: TOD;
		Break1_StartTime: TOD;
		Break1_EndTime: TOD;
		Break2_StartTime: TOD;
		Break2_EndTime: TOD;
		Break3_StartTime: TOD;
		Break3_EndTime: TOD;
		Shift_EndTime: TOD;
	END_STRUCT
END_TYPE

// ---- Data types/Generic udts/udt_Generic_ShiftConfigUDINT_20160531.TcDUT
(*udt (user defined type) for production shift config data In UDINT (Unsigned Double Integer) Format

	Author(S): Brent Lekx-Toniolo ;
	20160531:
		- Initial Concept
	
 


*)

TYPE udt_Generic_ShiftConfigUDINT_20160531 :
	STRUCT
		Shift_StartTime: UDINT;
		Break1_StartTime: UDINT;
		Break1_EndTime: UDINT;
		Break2_StartTime: UDINT;
		Break2_EndTime: UDINT;
		Break3_StartTime: UDINT;
		Break3_EndTime: UDINT;
		Shift_EndTime: UDINT;
	END_STRUCT
END_TYPE

// ---- Data types/Generic udts/udt_Generic_ShiftConfig_20160519.TcDUT
(*udt (user defined type) for production shift config data

	Author(S): Brent Lekx-Toniolo ;
	20160519:
		- Initial Concept
	


*)


TYPE udt_Generic_ShiftConfig_20160519 :
	STRUCT
		Shift_StartTime: OTSTRUCT;
		Break1_StartTime: OTSTRUCT;
		Break1_EndTime: OTSTRUCT;
		Break2_StartTime: OTSTRUCT;
		Break2_EndTime: OTSTRUCT;
		Break3_StartTime: OTSTRUCT;
		Break3_EndTime: OTSTRUCT;
		Shift_EndTime: OTSTRUCT;
	END_STRUCT
END_TYPE

// ---- Data types/Generic udts/udt_IVxx_Input_Image_20250812.TcDUT
(*udt (user defined type) for all fixture input interface
	auth. R.Jones of Sodecia GTAC

------------------------------------------------------------------------
REVISION NOTES:
	V1.0 
	- initial concept, r.jones *)
	
TYPE udt_IVxx_Input_Image_20250812 :
STRUCT
	IVx_Release: BOOL;
	FailureRecovery_Attempt_Max: INT;
	FailureRecovery_Enable: BOOL;
	IVx_Bypass: BOOL;
END_STRUCT
END_TYPE

// ---- Data types/Graco udts/udt_Graco_Input.TcDUT
(*udt (user defined type) of Graco Profibus Based Stud:
	auth.  Sodecia GTAC; 
	May 2013; version 1.0
	July 2020 Updated for new Graco GSD - j.vandongen
	*)

TYPE udt_Graco_Input :
	STRUCT
		(*Status Of Profibus Slave*)
		Inputs:udt_ProfiNode_Status;

		(*Input Bytes*)
		Byte0: BYTE;
		Byte1: BYTE;
		Byte2: BYTE;
		Byte3: BYTE;
		Byte4: BYTE;
		Byte5: BYTE;
		Byte6: BYTE;
		Byte7: BYTE;
		Byte8: BYTE;
		Byte9: BYTE;
		Byte10: BYTE;
		Byte11: BYTE;
		Byte12: BYTE;
		Byte13: BYTE;
		Byte14: BYTE;
		Byte15: BYTE;
		Byte16: BYTE;
		Byte17: BYTE;
		Byte18: BYTE;
		Byte19: BYTE;
		Byte20: BYTE;
		Byte21: BYTE;
		Byte22: BYTE;
		Byte23: BYTE;
		Byte24: BYTE;
		Byte25: BYTE;
		Byte26: BYTE;
		Byte27: BYTE;
		Byte28: BYTE;
		Byte29: BYTE;
		Byte30: BYTE;
		Byte31: BYTE;
		Byte32: BYTE;
		Byte33: BYTE;
		Byte34: BYTE;
		Byte35: BYTE;
		Byte36: BYTE;
		Byte37: BYTE;
		Byte38: BYTE;
		Byte39: BYTE;
		Byte40: BYTE;
		Byte41: BYTE;
		Byte42: BYTE;
		Byte43: BYTE;
		Byte44: BYTE;
		Byte45: BYTE;
		Byte46: BYTE;
		Byte47: BYTE;
		Byte48: BYTE;
		Byte49: BYTE;
		Byte50: BYTE;
		Byte51: BYTE;
		Byte52: BYTE;
		Byte53: BYTE;
		Byte54: BYTE;
		Byte55: BYTE;
		Byte56: BYTE;
		Byte57: BYTE;
		Byte58: BYTE;
		Byte59: BYTE;
		Byte60: BYTE;
		Byte61: BYTE;
		Byte62: BYTE;
		Byte63: BYTE;
		Byte64: BYTE;
		Byte65: BYTE;
		Byte66: BYTE;
		Byte67: BYTE;
		Byte68: BYTE;
		Byte69: BYTE;
		Byte70: BYTE;
		Byte71: BYTE;
		Byte72: BYTE;
		Byte73: BYTE;
		Byte74: BYTE;
		Byte75: BYTE;
		Byte76: BYTE;
		Byte77: BYTE;

	END_STRUCT
END_TYPE

// ---- Data types/Graco udts/udt_Graco_Outputs.TcDUT
(*udt (user defined type) of Graco Profibus Based Stud:
	auth.  Sodecia GTAC; 
	May 2013; version 1.0
	July 2020 Updated for new Graco GSD - j.vandongen
	*)


TYPE udt_Graco_Outputs :
	STRUCT

		Byte0: BYTE;
		Byte1: BYTE;
		Byte2: BYTE;
		Byte3: BYTE;
		Byte4: BYTE;
		Byte5: BYTE;
		Byte6: BYTE;
		Byte7: BYTE;
		Byte8: BYTE;
		Byte9: BYTE;
		Byte10: BYTE;
		Byte11: BYTE;
		Byte12: BYTE;
		Byte13: BYTE;
		Byte14: BYTE;
		Byte15: BYTE;
		Byte16: BYTE;
		Byte17: BYTE;
		Byte18: BYTE;
		Byte19: BYTE;
		Byte20: BYTE;
		Byte21: BYTE;
		Byte22: BYTE;
		Byte23: BYTE;
		Byte24: BYTE;
		Byte25: BYTE;
		Byte26: BYTE;
		Byte27: BYTE;
		Byte28: BYTE;
		Byte29: BYTE;
		Byte30: BYTE;
		Byte31: BYTE;

	END_STRUCT
END_TYPE

// ---- Data types/HardwareDiags/E_State.TcDUT
{attribute 'qualified_only'}
{attribute 'strict'}
//** = simply adjust these lines if modifying code for own purposes
 
// central declaration of state machine states 
// (supports easy program modification)
 
TYPE E_State :
(
    eState_InitiateStateMachine    		:= 0,     // initiate state machine (set parameters)
    eState_ReadTCatMajorVerInit       	:= 20,    //** initiate reading Twincat Major Version Number
    eState_ReadTCatMajorVer    			:= 21,    //** process reading Twincat Major Version Number
	eState_ReadTCatMinorVerInit   		:= 22,    //** initiate reading Twincat Minor Version Number
    eState_ReadTCatMinorVerTemp       	:= 23,    //** process reading Twincat Minor Version Number
	eState_ReadCPUTempInit        		:= 24,    //** initiate reading CPU Temperature
    eState_ReadCpuTemp		   			:= 25,    //** process reading CPU Temperature
	eState_ReadFanSpeedInit         	:= 26,    //** initiate reading Fan Speed
    eState_ReadFanSpeed			   		:= 27,    //** process reading Fan Speed
	eState_ReadMBoardTempInit        	:= 28,    //** initiate reading Motherboard Temperature
    eState_ReadMboardTemp			   	:= 29,    //** process reading Motherboard Temperature
    eState_ReadMBoardBootCountInit    	:= 30,    //** initiate reading Motherboard Boot Count
    eState_ReadMboardBootCount     		:= 31,    //** process reading Motherboard Boot Count
	eState_ReadMboardOpMinsInit   		:= 32,    //** initiate reading Motherboard Operational Time
    eState_ReadMboardOpMins       		:= 33,    //** process reading Motherboard Operational Time
	eState_Read5VSupplyInit        		:= 34,    //** initiate reading 5V Supply Voltage
    eState_Read5VSupply		   			:= 35,    //** process reading 5V Supply Voltage
	eState_Read12VSupplyInit         	:= 36,    //** initiate reading 12V Supply Voltage
    eState_Read12VSupply			   	:= 37,    //** process reading 12V Supply Voltage
	eState_ReadBattStatusInit        	:= 38,    //** initiate reading Battery Status
    eState_ReadBattStatus			   	:= 39,    //** process reading Battery Status
	eState_ReadBattReplaceDateInit    	:= 40,    //** initiate reading Battery Replacement Date
    eState_ReadBattReplaceDate		   	:= 41,    //** process reading Battery Replacement Date
	eState_ReadBattCapcityInit         	:= 42,    //** initiate reading Battery Capacity
    eState_ReadBattCapacity        		:= 43,    //** initiate reading Battery Capacity
	eState_ReadBattRuntimeInit        	:= 44,    //** initiate reading Battery Runtime 
    eState_ReadBattRuntime			   	:= 45,    //** process reading Battery Runtime	
    eState_IdleState               		:= 100    // idle state 
) UINT;
END_TYPE

// ---- Data types/HardwareDiags/udt_HardwareDiags.TcDUT
TYPE udt_HardwareDiags :
STRUCT
	TwinCATMajorRev: 		UINT;
	TwinCATMinorRev: 		UINT;
	TwinCATRevision: 		STRING;
	CpuTemp: 				INT;
	FanSpeed:			 	INT;
	MboardTemp:				INT;
	BootCount:				DINT;
	OpTime:					DINT;
	Supply5V:				INT;
	Supply12V:				INT;
	BatteryStatus:			BYTE;
	BatteryReplaceDate:		STRING;
	BatteryCapacity:		BYTE;
	BatteryRuntime:			DINT;		
END_STRUCT
END_TYPE

// ---- Data types/Keyence/udt_IV2_DiscreteImage.TcDUT
TYPE udt_IV2_DiscreteImage :
STRUCT
	ProgramNumber:INT;
	TriggerOutput:BOOL;
	ErrorStatus:BOOL;
	ErrorCode:UINT;
	Running:BOOL;
	Busy:BOOL;
	TriggerReady:BOOL;
	InfoData:udt_ECATSlave_Status;
	ResultAvailable:BOOL;
	OverallJudgementOK:BOOL;
	TriggerResponse:BOOL;
	TriggerFailed:BOOL;
	PortB_MissingLink: BOOL;
	Faulted: BOOL;
	
	IV_Check_OK : BOOL;
	IV_Check_NOK : BOOL;	
	
	Fault_Failure_Recovery : ARRAY[1..15] OF BOOL;
	Failure_Max_Attempt_Fault : BOOL;
		
END_STRUCT
END_TYPE

// ---- Data types/Keyence/udt_IV2_Inputs.TcDUT
TYPE udt_IV2_Inputs :
STRUCT
	Error_Status:BOOL;
	ErrorCode:UINT;
	PositionAdjMatch:DINT;
	ToolMatch:ARRAY [1..13] OF DINT;
	ToolResult:ARRAY[1..13] OF BOOL;
	ProgramSwitchOK:BOOL;
	ProgramSwitchFailed:BOOL;
	ResultAvailable:BOOL;
	OverallJudgementOK:BOOL;
	ProgramNumber:INT;
	TriggerResponse:BOOL;
	TriggerFailed:BOOL;
	ResultUpdateComplete:BOOL;
	PositionCorrectionStatus:BOOL;
	MasterRegResponse:BOOL;
	MasterRegFailed:BOOL;
	SDCardStopResponse:BOOL;
	SDCardStopFailed:BOOL;
	LogicResult:ARRAY[1..4] OF BOOL;
	StatsResetResponse:BOOL;
	Running:BOOL;
	ErrorClearResponse:BOOL;
	Busy:BOOL;
	TriggerReady:BOOL;
	NoFreeSpaceSD:BOOL;
	InfoData:udt_ECATSlave_Status;
END_STRUCT
END_TYPE

// ---- Data types/Keyence/udt_IV2_Outputs.TcDUT
TYPE udt_IV2_Outputs :
STRUCT
	Program_Switch_RQST:BOOL;
	Trigger_RQST:BOOL;
	Master_Image_RQST:BOOL;
	SD_Save_Stop_RQST:BOOL;
	Reset_Statistics_RQST:BOOL;
	Error_Clear_RQST:BOOL;
	ProgramNum:ARRAY[0..3] OF BOOL;
END_STRUCT
END_TYPE

// ---- Data types/Robot_udts/udt_EtherCAT_Kuka_InputBits_20121204.TcDUT
(*udt (user defined type) for all KUKA KRC4 Robot systems on EL6692 ECAT Bridge
	Author(S): Brent Lekx-Toniolo of Sodecia GTAC;
	Version 1.0: November 2012
		- Initial Concept
	Version 20121204
		Changes from v1
			- Change to Naming Convention to include date as version

	Last Edit: December 4th, 2012, blt
*)
TYPE udt_EtherCAT_Kuka_InputBits_20121204 :
STRUCT
	Robot_OUT: ARRAY [1..512] OF BOOL;
END_STRUCT
END_TYPE

// ---- Data types/Robot_udts/udt_EtherCAT_Kuka_OutputBits_20121204.TcDUT
(*udt (user defined type) for all KUKA KRC4 Robot systems on EL6692 ECAT Bridge
	Author(S): Brent Lekx-Toniolo of Sodecia GTAC;
	Version 1.0: November 2012
		- Initial Concept
	Version 20121204
		Changes from v1
			- Change to Naming Convention to include date as version

	Last Edit: December 4th, 2012, blt
*)
TYPE udt_EtherCAT_Kuka_OutputBits_20121204 :
STRUCT
	Robot_IN: ARRAY [1..512] OF BOOL;
END_STRUCT
END_TYPE

// ---- Data types/Robot_udts/udt_EtherCAT_Motoman_Input_20151105.TcDUT
(*udt (user defined type) for all Motoman Robot Controllers with HMS AnyBus Profibus Interface Card
	Author(S): Brent Lekx-Toniolo/Rob Remillard of Sodecia GTAC;
	Version 1.0: August 2010
		- Initial Concept
	Version 20121204
		Changes from v1
			- Increased Size to 32 Bytes
			- Change to Naming Convention to include date as version

	Last Edit: December 4th, 2012, blt
*)

TYPE udt_EtherCAT_Motoman_Input_20151105 :
	STRUCT
	InfoData: udt_ECATSlave_Status;
		(*Output Data From Robot, 32 Bytes total size*)
		SYS:UDINT;
		OG4: BYTE;
		OG5: BYTE;
		OG6: BYTE;
		OG7: BYTE;
		OG8: BYTE;
		OG9: BYTE;
		OG10: BYTE;
		OG11: BYTE;
		OG12: BYTE;
		OG13: BYTE;
		OG14: BYTE;
		OG15: BYTE;
		OG16: BYTE;
		OG17: BYTE;
		OG18: BYTE;
		OG19: BYTE;
		OG20: BYTE;
		OG21: BYTE;
		OG22: BYTE;
		OG23: BYTE;
		OG24: BYTE;
		OG25: BYTE;
		OG26: BYTE;
		OG27: BYTE;
		OG28: BYTE;
		OG29: BYTE;
		OG30: BYTE;
		OG31: BYTE;
		OG32: BYTE;
		OG33: BYTE;
	END_STRUCT
END_TYPE

// ---- Data types/Robot_udts/udt_EtherCAT_Motoman_Output_20151105.TcDUT
(*udt (user defined type) for all Motoman Robot Controllers with HMS AnyBus Profibus Interface Card
	Author(S): Brent Lekx-Toniolo/Rob Remillard of Sodecia GTAC;
	Version 1.0: August 2010
		- Initial Concept
	Version 20121204
		Changes from v1
			- Increased Size to 32 Bytes
			- Change to Naming Convention to include date as version

	Last Edit: December 4th, 2012, blt
*)
TYPE udt_EtherCAT_Motoman_Output_20151105 :
	STRUCT
		(*Input Data To Robot, 32 Bytes total size*)
		SYS:UDINT;
		IG4:BYTE;
		IG5:BYTE;
		IG6:BYTE;
		IG7:BYTE;
		IG8:BYTE;
		IG9:BYTE;
		IG10:BYTE;
		IG11:BYTE;
		IG12:BYTE;
		IG13:BYTE;
		IG14:BYTE;
		IG15:BYTE;
		IG16:BYTE;
		IG17:BYTE;
		IG18:BYTE;
		IG19:BYTE;
		IG20:BYTE;
		IG21:BYTE;
		IG22:BYTE;
		IG23:BYTE;
		IG24:BYTE;
		IG25:BYTE;
		IG26:BYTE;
		IG27:BYTE;
		IG28:BYTE;
		IG29:BYTE;
		IG30:BYTE;
		IG31:BYTE;
		IG32:BYTE;
		IG33:BYTE;
		END_STRUCT
END_TYPE

// ---- Data types/Robot_udts/udt_GenericRobot_AnyFieldbus_Input58Bytes.TcDUT
(*udt (user defined type) for all Fieldbus Based Robot Interfacing Template for 58 bytes
	Author(S): Brent Lekx-Toniolo of Sodecia GTAC;
	Version 1.0: March 2013
		- Initial Concept
	Version 20130319

	Last Edit: March 19th, 2013, blt
*)
TYPE udt_GenericRobot_AnyFieldbus_Input58Bytes :
STRUCT
	BYTE_: ARRAY [1..58] OF BYTE;
END_STRUCT
END_TYPE

// ---- Data types/Robot_udts/udt_GenericRobot_AnyFieldbus_InputBytes_20220421.TcDUT
(*udt (user defined type) for all Fieldbus Based Robot Interfacing up to 64 Bytes
	Author(S): Brent Lekx-Toniolo of Sodecia GTAC;
	Version 1.0: November 2012
		- Initial Concept
	Version 20121204
		Changes from v1
			- Change to Naming Convention to include date as version
	Version 20220421
			- Changed starting point of Array fro 1 to 0 for TcHmi conventions, b.lekx-toniolo
*)
TYPE udt_GenericRobot_AnyFieldbus_InputBytes_20220421 :
STRUCT
	BYTE_: ARRAY [0..64] OF BYTE;
END_STRUCT
END_TYPE

// ---- Data types/Robot_udts/udt_GenericRobot_AnyFieldbus_Output58Bytes.TcDUT
(*udt (user defined type) for all Fieldbus Based Robot Interfacing Template for 58 bytes
	Author(S): Brent Lekx-Toniolo of Sodecia GTAC;
	Version 1.0: March 2013
		- Initial Concept
	Version 20130319

	Last Edit: March 19th, 2013, blt
*)

TYPE udt_GenericRobot_AnyFieldbus_Output58Bytes :
STRUCT
	Byte_: ARRAY [1..58] OF BYTE;
END_STRUCT
END_TYPE

